C04750=3783,34311,-25890,658,-28447,-2203
C04751=3764,34294,-25911,661,-28441,-2195
C04752=3742,34281,-25927,664,-28436,-2187
C04753=3760,34297,-25907,662,-28442,-2194
C04754=3779,34307,-25895,659,-28446,-2201
C04755=3789,34330,-25867,657,-28455,-2205
C04756=3806,34351,-25841,655,-28463,-2211
C04757=3823,34373,-25815,652,-28471,-2218
C04758=3840,34394,-25789,650,-28479,-2225
C04759=3857,34415,-25763,647,-28487,-2231
C04760=3874,34437,-25737,645,-28495,-2238
C04761=3889,34459,-25710,642,-28504,-2243
C04762=3900,34481,-25683,641,-28512,-2248
C04763=3910,34504,-25655,639,-28521,-2251
C04764=3920,34527,-25627,637,-28530,-2255
C04765=3929,34550,-25599,636,-28538,-2259
C04766=3939,34574,-25571,634,-28547,-2263
C04767=3949,34597,-25543,633,-28556,-2266
C04768=3958,34620,-25514,631,-28565,-2270
C04769=3955,34646,-25483,632,-28574,-2269
C04770=3962,34670,-25454,630,-28583,-2271
C04771=3970,34693,-25425,629,-28592,-2274
C04772=3969,34719,-25394,629,-28602,-2273
C04773=3974,34743,-25364,628,-28611,-2275
C04774=3971,34770,-25333,628,-28621,-2274
C04775=3968,34796,-25301,629,-28630,-2273
C04776=3965,34822,-25269,629,-28640,-2271
C04777=3956,34845,-25241,630,-28648,-2268
C04778=3948,34868,-25213,631,-28657,-2265
C04779=3938,34890,-25187,632,-28665,-2260
C04780=3925,34911,-25162,634,-28673,-2255
C04781=3913,34932,-25137,635,-28680,-2251
C04782=3920,34941,-25125,634,-28684,-2253
C04783=3935,34922,-25149,632,-28677,-2259
C04784=3946,34901,-25174,631,-28669,-2264
C04785=3958,34880,-25200,629,-28661,-2268
C04786=3970,34859,-25225,628,-28654,-2273
C04787=3973,34832,-25257,628,-28644,-2275
C04788=3985,34812,-25282,626,-28636,-2279
C04789=3988,34785,-25313,626,-28627,-2281
C04790=3991,34759,-25345,626,-28617,-2282
C04791=3984,34735,-25374,627,-28608,-2279
C04792=3987,34709,-25406,627,-28598,-2281
C04793=3987,34709,-24006,627,-28598,-2281
C04794=3534,35026,-21027,687,-28710,-2102
C04795=3534,35026,-25027,687,-28710,-2102
C04796=3539,35031,-25020,687,-28712,-2103
C04797=3543,35037,-25013,686,-28714,-2105
C04798=3542,35044,-25005,686,-28717,-2105
C04799=3545,35050,-24998,686,-28719,-2106
C04800=3549,35055,-24991,685,-28721,-2107
C04801=3554,35061,-24984,684,-28724,-2109
C04802=3558,35067,-24977,684,-28726,-2111
C04803=3565,35069,-24975,683,-28727,-2113
C04804=3571,35071,-24971,682,-28728,-2115
C04805=3575,35077,-24964,681,-28730,-2117
C04806=3579,35083,-24958,681,-28732,-2119
C04807=3584,35088,-24951,680,-28734,-2121
C04808=3589,35091,-24947,679,-28735,-2123
C04809=3596,35092,-24946,678,-28736,-2125
C04810=3603,35093,-24944,677,-28736,-2128
C04811=3610,35095,-24943,676,-28737,-2131
C04812=3616,35097,-24939,675,-28738,-2133
C04813=3621,35103,-24932,675,-28740,-2135
C04814=3620,35108,-24927,675,-28742,-2135
C04815=3615,35112,-24922,675,-28743,-2133
C04816=3609,35116,-24917,676,-28745,-2130
C04817=3604,35120,-24912,677,-28746,-2128
C04818=3598,35121,-24911,678,-28747,-2126
C04819=3591,35120,-24912,679,-28746,-2123
C04820=3584,35119,-24913,680,-28746,-2120
C04821=3577,35118,-24914,681,-28745,-2118
C04822=3570,35117,-24916,682,-28745,-2115
C04823=3563,35116,-24917,683,-28744,-2112
C04824=3556,35115,-24918,684,-28744,-2109
C04825=3549,35114,-24920,685,-28743,-2107
C04826=3542,35113,-24921,686,-28743,-2104
C04827=3535,35112,-24922,687,-28742,-2101
C04828=3528,35111,-24924,688,-28742,-2099
C04829=3521,35110,-24925,689,-28741,-2096
C04830=3515,35108,-24928,689,-28740,-2093
C04831=3511,35102,-24935,690,-28738,-2092
C04832=3505,35098,-24940,691,-28737,-2090
C04833=3498,35097,-24941,692,-28736,-2087
C04834=3491,35096,-24942,693,-28736,-2084
C04835=3484,35095,-24944,694,-28735,-2082
C04836=3477,35094,-24945,695,-28735,-2079
C04837=3471,35093,-24946,696,-28734,-2076
C04838=3466,35088,-24952,696,-28732,-2074
C04839=3461,35082,-24959,697,-28730,-2073
C04840=3462,35076,-24967,697,-28728,-2073
C04841=3462,35069,-24976,697,-28725,-2073
C04842=3463,35062,-24984,697,-28723,-2073
C04843=3464,35055,-24992,697,-28720,-2074
C04844=3468,35050,-24998,696,-28719,-2075
C04845=3474,35046,-25003,696,-28717,-2078
C04846=3479,35042,-25008,695,-28716,-2080
C04847=3485,35038,-25013,694,-28714,-2082
C04848=3490,35034,-25018,693,-28713,-2084
C04849=3496,35030,-25023,693,-28711,-2086
C04850=3501,35026,-25028,692,-28710,-2088
C04851=3507,35022,-25032,691,-28708,-2091
C04852=3514,35023,-25031,690,-28709,-2093
C04853=3520,35024,-25029,689,-28709,-2096
C04854=3527,35025,-25028,688,-28710,-2099
C04855=3534,35026,-25027,687,-28710,-2102
C04856=3534,35026,-23627,687,-28710,-2102
C04857=3901,34041,-22216,644,-28348,-2250
C04858=3901,34041,-26216,644,-28348,-2250
C04859=3933,34017,-26245,639,-28340,-2263
C04860=3959,33989,-26278,636,-28330,-2273
C04861=3985,33961,-26312,632,-28319,-2284
C04862=4016,33935,-26343,628,-28310,-2296
C04863=4038,33905,-26380,626,-28299,-2304
C04864=4064,33877,-26413,622,-28289,-2315
C04865=4090,33849,-26447,619,-28279,-2325
C04866=4116,33821,-26481,615,-28269,-2336
C04867=4136,33789,-26519,613,-28257,-2343
C04868=4162,33761,-26553,609,-28247,-2354
C04869=4187,33732,-26588,606,-28237,-2364
C04870=4210,33702,-26623,603,-28226,-2373
C04871=4234,33673,-26659,599,-28215,-2382
C04872=4257,33643,-26695,597,-28204,-2391
C04873=4281,33613,-26731,593,-28193,-2401
C04874=4300,33582,-26769,591,-28182,-2409
C04875=4320,33550,-26807,588,-28170,-2417
C04876=4341,33518,-26845,586,-28159,-2425
C04877=4364,33489,-26881,582,-28148,-2434
C04878=4386,33458,-26918,579,-28137,-2443
C04879=4406,33426,-26956,577,-28125,-2451
C04880=4425,33394,-26995,574,-28113,-2458
C04881=4446,33363,-27033,572,-28102,-2467
C04882=4462,33329,-27074,570,-28089,-2473
C04883=4486,33299,-27110,566,-28079,-2482
C04884=4500,33264,-27152,565,-28066,-2488
C04885=4519,33232,-27191,562,-28054,-2496
C04886=4538,33199,-27230,560,-28042,-2503
C04887=4553,33165,-27272,558,-28029,-2509
C04888=4555,33137,-27306,558,-28019,-2510
C04889=4535,33169,-27267,560,-28031,-2502
C04890=4517,33202,-27227,563,-28043,-2495
C04891=4502,33236,-27186,565,-28055,-2489
C04892=4480,33267,-27149,568,-28066,-2480
C04893=4456,33297,-27113,571,-28077,-2471
C04894=4442,33332,-27071,573,-28090,-2465
C04895=4419,33361,-27035,576,-28101,-2456
C04896=4395,33391,-26999,579,-28112,-2447
C04897=4381,33426,-26956,580,-28125,-2441
C04898=4358,33456,-25521,584,-28136,-2432
C04899=-41004,59868,4099,4900,-34257,16705
C04900=-41004,59868,1099,4900,-34257,16705
C04901=-41004,64596,1380,5213,-31659,16463
C04902=-41004,59868,1099,4900,-34257,16705
C04903=-41004,59868,9099,4900,-34257,16705
C04904=4358,33456,-22921,584,-28136,-2432
C04905=4358,33456,-26921,584,-28136,-2432
C04906=4336,33487,-26884,586,-28147,-2423
C04907=4316,33518,-26845,589,-28158,-2415
C04908=4296,33550,-26807,592,-28170,-2407
C04909=4274,33581,-26771,595,-28181,-2398
C04910=4251,33610,-26735,598,-28192,-2389
C04911=4230,33642,-26697,600,-28203,-2381
C04912=4204,33670,-26663,604,-28214,-2371
C04913=4184,33702,-26625,606,-28225,-2363
C04914=4158,33730,-26591,610,-28235,-2352
C04915=4135,33759,-26555,613,-28246,-2343
C04916=4112,33789,-26519,616,-28257,-2334
C04917=4088,33819,-26483,619,-28268,-2325
C04918=4065,33849,-26447,622,-28279,-2315
C04919=4040,33877,-26413,625,-28289,-2305
C04920=4014,33905,-26379,629,-28299,-2295
C04921=3988,33933,-26346,632,-28309,-2285
C04922=3962,33961,-26312,636,-28319,-2274
C04923=3935,33990,-26278,639,-28330,-2264
C04924=3909,34018,-26244,643,-28340,-2254
C04925=3901,34041,-26216,644,-28348,-2250
C04926=3901,34041,-24816,644,-28348,-2250
C04927=3701,33792,-22519,674,-28253,-2173
C04928=3701,33792,-26519,674,-28253,-2173
C04929=3740,33763,-26554,669,-28243,-2189
C04930=3773,33730,-26594,664,-28231,-2202
C04931=3812,33701,-26629,659,-28221,-2217
C04932=3839,33664,-26673,655,-28207,-2228
C04933=3871,33631,-26713,651,-28195,-2241
C04934=3897,33594,-26757,648,-28182,-2251
C04935=3929,33561,-26798,644,-28170,-2264
C04936=3957,33524,-26841,640,-28157,-2275
C04937=3983,33488,-26885,636,-28143,-2285
C04938=4009,33451,-26930,633,-28130,-2296
C04939=4035,33414,-26975,630,-28116,-2306
C04940=4062,33377,-27018,626,-28103,-2317
C04941=4089,33341,-27063,623,-28090,-2327
C04942=4109,33300,-27112,620,-28075,-2335
C04943=4135,33263,-27156,617,-28061,-2346
C04944=4156,33223,-27204,614,-28047,-2354
C04945=4180,33185,-27250,611,-28033,-2364
C04946=4204,33147,-27296,608,-28019,-2373
C04947=4229,33109,-27342,604,-28005,-2383
C04948=4255,33072,-27387,601,-27991,-2393
C04949=4282,33035,-27431,597,-27978,-2404
C04950=4308,32999,-27475,594,-27965,-2415
C04951=4335,32962,-27520,590,-27951,-2425
C04952=4362,32925,-27564,587,-27938,-2436
C04953=4389,32888,-27608,583,-27924,-2446
C04954=4415,32852,-27652,580,-27911,-2457
C04955=4442,32815,-27697,576,-27898,-2468
C04956=4462,32774,-27746,574,-27883,-2476
C04957=4461,32750,-27775,574,-27874,-2475
C04958=4436,32788,-27730,577,-27888,-2465
C04959=4412,32826,-27684,580,-27901,-2456
C04960=4387,32864,-27638,584,-27915,-2446
C04961=4360,32901,-27594,587,-27929,-2435
C04962=4333,32937,-27549,591,-27942,-2425
C04963=4304,32973,-27507,595,-27955,-2413
C04964=4280,33011,-27461,598,-27969,-2403
C04965=4253,33048,-27416,601,-27982,-2393
C04966=4226,33084,-27372,605,-27996,-2382
C04967=4200,33121,-27328,608,-28009,-2372
C04968=4173,33158,-27284,612,-28022,-2361
C04969=4153,33198,-27235,615,-28037,-2353
C04970=4127,33235,-27190,618,-28051,-2343
C04971=4107,33276,-27141,621,-28066,-2335
C04972=4080,33312,-27097,624,-28079,-2324
C04973=4060,33353,-27048,627,-28094,-2316
C04974=4034,33390,-27004,630,-28107,-2306
C04975=4004,33424,-26962,634,-28120,-2294
C04976=3980,33462,-26916,637,-28134,-2284
C04977=3955,33500,-26871,640,-28147,-2274
C04978=3922,33533,-26831,645,-28159,-2261
C04979=3896,33570,-26787,648,-28173,-2251
C04980=3865,33604,-26746,652,-28185,-2239
C04981=3836,33639,-26703,656,-28198,-2227
C04982=3808,33675,-26660,660,-28211,-2216
C04983=3775,33708,-26621,664,-28223,-2203
C04984=3738,33739,-26584,669,-28234,-2188
C04985=3699,33768,-26549,674,-28244,-2173
C04986=3660,33797,-26514,680,-28255,-2157
C04987=3658,33810,-26499,680,-28259,-2157
C04988=3701,33792,-26519,674,-28253,-2173
C04989=3701,33792,-25119,674,-28253,-2173
C04990=3330,33582,-22776,728,-28171,-2030
C04991=3330,33582,-26776,728,-28171,-2030
C04992=3394,33535,-26833,719,-28154,-2055
C04993=3460,33494,-26882,710,-28140,-2081
C04994=3517,33443,-26944,703,-28121,-2104
C04995=3581,33396,-27001,694,-28104,-2129
C04996=3635,33342,-27064,687,-28085,-2150
C04997=3690,33289,-27128,680,-28066,-2172
C04998=3740,33234,-27195,673,-28046,-2192
C04999=3785,33175,-27266,667,-28025,-2210
C05000=3829,33116,-27336,661,-28003,-2227
C05001=3875,33058,-27407,655,-27982,-2245
C05002=3921,33000,-27476,649,-27961,-2264
C05003=3968,32942,-27546,643,-27940,-2282
C05004=4014,32884,-27616,637,-27919,-2301
C05005=4060,32826,-27686,631,-27898,-2319
C05006=4098,32764,-27762,626,-27875,-2334
C05007=4144,32706,-27832,620,-27854,-2352
C05008=4188,32646,-27903,614,-27832,-2370
C05009=4233,32587,-27974,608,-27811,-2388
C05010=4275,32527,-28047,602,-27788,-2404
C05011=4322,32469,-28117,596,-27767,-2423
C05012=4362,32407,-28191,591,-27745,-2439
C05013=4408,32349,-28262,585,-27723,-2457
C05014=4454,32290,-28333,578,-27702,-2475
C05015=4506,32235,-28399,571,-27682,-2495
C05016=4558,32180,-28466,564,-27662,-2516
C05017=4611,32125,-28532,557,-27642,-2537
C05018=4663,32070,-28598,550,-27622,-2557
C05019=4716,32015,-28664,543,-27602,-2578
C05020=4775,31964,-28725,535,-27584,-2601
C05021=4803,31910,-28791,531,-27564,-2613
C05022=4751,31965,-28725,538,-27584,-2592
C05023=4691,32016,-28664,546,-27602,-2569
C05024=4639,32071,-28597,553,-27622,-2548
C05025=4586,32125,-28531,561,-27642,-2527
C05026=4528,32177,-28469,569,-27661,-2504
C05027=4480,32235,-28399,575,-27682,-2486
C05028=4429,32290,-28333,582,-27702,-2465
C05029=4383,32349,-28262,588,-27723,-2447
C05030=4339,32408,-28190,594,-27745,-2430
C05031=4293,32466,-28120,600,-27766,-2411
C05032=4254,32529,-28045,605,-27789,-2396
C05033=4208,32587,-27975,611,-27810,-2378
C05034=4164,32646,-27903,617,-27832,-2360
C05035=4119,32705,-27832,623,-27853,-2342
C05036=4077,32766,-27759,629,-27876,-2326
C05037=4031,32824,-27689,635,-27897,-2307
C05038=3984,32882,-27619,641,-27918,-2289
C05039=3939,32940,-27549,647,-27939,-2271
C05040=3901,33003,-27473,652,-27962,-2256
C05041=3855,33061,-27404,658,-27983,-2237
C05042=3809,33119,-27334,664,-28004,-2219
C05043=3761,33176,-27265,670,-28025,-2200
C05044=3716,33234,-27194,676,-28046,-2183
C05045=3661,33287,-27131,684,-28065,-2161
C05046=3608,33341,-27067,691,-28084,-2140
C05047=3551,33392,-27005,698,-28103,-2117
C05048=3493,33444,-26943,706,-28121,-2094
C05049=3429,33491,-26886,715,-28138,-2069
C05050=3366,33539,-26829,723,-28155,-2044
C05051=3330,33582,-26776,728,-28171,-2030
C05052=3330,33582,-25376,728,-28171,-2030
C05053=3223,32799,-23726,750,-27878,-1993
C05054=3223,32799,-27726,750,-27878,-1993
C05055=3252,32786,-27741,746,-27874,-2004
C05056=3276,32766,-27765,743,-27867,-2014
C05057=3297,32744,-27792,740,-27859,-2022
C05058=3323,32724,-27815,737,-27852,-2032
C05059=3350,32705,-27838,733,-27845,-2043
C05060=3374,32685,-27862,730,-27838,-2052
C05061=3395,32663,-27889,727,-27830,-2061
C05062=3422,32643,-27913,723,-27823,-2071
C05063=3448,32624,-27936,720,-27816,-2081
C05064=3468,32601,-27964,717,-27808,-2089
C05065=3494,32581,-27987,714,-27801,-2100
C05066=3520,32562,-28010,710,-27794,-2110
C05067=3540,32539,-28038,707,-27785,-2118
C05068=3566,32519,-28061,704,-27778,-2128
C05069=3593,32500,-28085,700,-27771,-2138
C05070=3619,32481,-28108,697,-27765,-2149
C05071=3639,32458,-28136,694,-27756,-2157
C05072=3665,32438,-28159,690,-27749,-2167
C05073=3691,32419,-28182,687,-27742,-2177
C05074=3718,32400,-26805,683,-27735,-2188
C05075=-41004,59868,4099,4900,-34257,16705
C05076=-41004,59868,1099,4900,-34257,16705
C05077=-41004,64596,1380,5213,-31659,16463
C05078=-41004,59868,1099,4900,-34257,16705
C05079=-41004,59868,9099,4900,-34257,16705
C05080=3718,32400,-24205,683,-27735,-2188
C05081=3718,32400,-28205,683,-27735,-2188
C05082=3744,32380,-28229,679,-27729,-2198
C05083=3771,32361,-28252,676,-27722,-2209
C05084=3797,32341,-28275,672,-27715,-2219
C05085=3817,32318,-28303,670,-27706,-2227
C05086=3844,32299,-28326,666,-27699,-2237
C05087=3872,32287,-28341,662,-27695,-2249
C05088=3899,32267,-28364,658,-27688,-2259
C05089=3926,32251,-28384,654,-27682,-2270
C05090=3954,32236,-28402,651,-27677,-2281
C05091=3946,32225,-28415,652,-27673,-2278
C05092=3918,32240,-28397,656,-27678,-2267
C05093=3890,32256,-28377,660,-27684,-2256
C05094=3861,32269,-28363,664,-27688,-2245
C05095=3835,32288,-28339,667,-27695,-2234
C05096=3808,32307,-28316,671,-27702,-2224
C05097=3784,32322,-28299,674,-27707,-2214
C05098=3760,32343,-28274,678,-27715,-2205
C05099=3733,32362,-28250,681,-27722,-2194
C05100=3707,32381,-28227,685,-27729,-2184
C05101=3680,32401,-28204,688,-27736,-2173
C05102=3654,32420,-28181,692,-27742,-2163
C05103=3628,32440,-28158,696,-27749,-2152
C05104=3601,32459,-28134,699,-27756,-2142
C05105=3582,32482,-28106,702,-27765,-2134
C05106=3555,32501,-28083,706,-27772,-2124
C05107=3529,32521,-28060,709,-27779,-2114
C05108=3502,32540,-28037,713,-27785,-2103
C05109=3483,32563,-28009,715,-27794,-2095
C05110=3457,32583,-27986,719,-27801,-2085
C05111=3437,32606,-27958,721,-27809,-2077
C05112=3411,32625,-27935,725,-27816,-2067
C05113=3384,32644,-27911,729,-27823,-2056
C05114=3365,32668,-27883,731,-27831,-2049
C05115=3339,32687,-27860,735,-27838,-2038
C05116=3312,32706,-27837,738,-27845,-2028
C05117=3293,32730,-27809,741,-27854,-2020
C05118=3267,32749,-27786,744,-27860,-2010
C05119=3246,32771,-27759,747,-27869,-2002
C05120=3221,32791,-27735,751,-27876,-1992
C05121=3223,32799,-27726,750,-27878,-1993
C05122=3223,32799,-26326,750,-27878,-1993
C05123=4368,32765,-23758,587,-27878,-2439
C05124=4368,32765,-27758,587,-27878,-2439
C05125=4392,32738,-27791,584,-27868,-2448
C05126=4406,32705,-27830,582,-27856,-2454
C05127=4423,32674,-27868,580,-27845,-2461
C05128=4441,32644,-27904,578,-27834,-2468
C05129=4457,32612,-27943,576,-27822,-2474
C05130=4477,32583,-27978,573,-27812,-2482
C05131=4495,32553,-28014,571,-27800,-2490
C05132=4517,32524,-28048,568,-27790,-2498
C05133=4538,32496,-28083,565,-27780,-2507
C05134=4556,32465,-28120,562,-27768,-2514
C05135=4578,32437,-28154,559,-27758,-2523
C05136=4600,32408,-28188,557,-27748,-2531
C05137=4618,32378,-28225,554,-27737,-2538
C05138=4639,32349,-28260,551,-27726,-2547
C05139=4661,32321,-28294,548,-27716,-2555
C05140=4679,32291,-28330,546,-27705,-2563
C05141=4700,32262,-28365,543,-27694,-2571
C05142=4723,32234,-28399,540,-27684,-2580
C05143=4741,32204,-28436,538,-27673,-2587
C05144=4761,32174,-28471,535,-27662,-2595
C05145=4784,32147,-28504,532,-27652,-2604
C05146=4803,32116,-28541,529,-27641,-2612
C05147=4823,32087,-28577,527,-27630,-2619
C05148=4846,32059,-28610,524,-27620,-2629
C05149=4860,32027,-28649,522,-27608,-2634
C05150=4883,31999,-28683,519,-27598,-2643
C05151=4898,31966,-28722,517,-27586,-2649
C05152=4920,31938,-28756,514,-27575,-2658
C05153=4936,31906,-28794,512,-27564,-2664
C05154=4950,31874,-28834,510,-27552,-2670
C05155=4927,31901,-28801,513,-27562,-2661
C05156=4912,31934,-28761,515,-27574,-2655
C05157=4889,31961,-28728,518,-27584,-2646
C05158=4870,31991,-28692,521,-27595,-2638
C05159=4851,32021,-28656,523,-27606,-2631
C05160=4827,32049,-28623,526,-27616,-2621
C05161=4808,32078,-28587,529,-27627,-2614
C05162=4789,32109,-28550,531,-27638,-2606
C05163=4766,32136,-28517,535,-27648,-2597
C05164=4746,32166,-28481,537,-27659,-2589
C05165=4728,32196,-28445,540,-27670,-2582
C05166=4705,32224,-28411,543,-27680,-2573
C05167=4684,32253,-28376,546,-27691,-2565
C05168=4666,32283,-28340,548,-27702,-2557
C05169=4644,32311,-28306,551,-27712,-2549
C05170=4623,32340,-28271,554,-27722,-2540
C05171=4604,32370,-28234,556,-27734,-2533
C05172=4583,32399,-28200,559,-27744,-2524
C05173=4561,32427,-28166,562,-27754,-2516
C05174=4543,32458,-28129,564,-27766,-2509
C05175=4522,32486,-28094,567,-27776,-2500
C05176=4500,32515,-28060,570,-27786,-2492
C05177=4482,32545,-28024,572,-27797,-2485
C05178=4461,32574,-27989,575,-27808,-2476
C05179=4439,32602,-27955,578,-27818,-2468
C05180=4424,32634,-27916,580,-27830,-2462
C05181=4409,32667,-27877,582,-27842,-2456
C05182=4391,32697,-27840,584,-27853,-2448
C05183=4373,32727,-27804,587,-27864,-2441
C05184=4368,32765,-27758,587,-27878,-2439
C05185=4368,32765,-26358,587,-27878,-2439
C05186=4624,32810,-23702,550,-27898,-2539
C05187=4624,32810,-27702,550,-27898,-2539
C05188=4618,32864,-27636,551,-27918,-2536
C05189=4611,32919,-27570,551,-27938,-2533
C05190=4605,32973,-27504,552,-27958,-2530
C05191=4598,33027,-27438,552,-27978,-2528
C05192=4592,33082,-27373,553,-27999,-2525
C05193=4604,33118,-27328,551,-28012,-2530
C05194=4623,33071,-27385,549,-27995,-2537
C05195=4630,33017,-27451,548,-27975,-2540
C05196=4636,32962,-27517,547,-27955,-2543
C05197=4643,32908,-27583,547,-27934,-2545
C05198=4649,32854,-27648,546,-27914,-2548
C05199=4665,32805,-27708,544,-27896,-2555
C05200=4680,32755,-27768,543,-27878,-2561
C05201=4688,32701,-27833,542,-27858,-2564
C05202=4710,32656,-27888,539,-27841,-2573
C05203=4729,32609,-27945,537,-27824,-2580
C05204=4747,32560,-28003,534,-27806,-2588
C05205=4770,32516,-28057,531,-27790,-2597
C05206=4796,32472,-28110,528,-27773,-2607
C05207=4822,32429,-28162,525,-27757,-2617
C05208=4847,32385,-28215,521,-27741,-2628
C05209=4879,32345,-28263,517,-27727,-2640
C05210=4904,32301,-28316,514,-27711,-2650
C05211=4930,32257,-28369,510,-27695,-2660
C05212=4959,32216,-28419,506,-27679,-2672
C05213=4987,32173,-28470,502,-27664,-2683
C05214=5019,32133,-28519,498,-27649,-2696
C05215=5046,32090,-28571,495,-27633,-2706
C05216=5072,32047,-28624,491,-27617,-2716
C05217=5102,32006,-28673,487,-27602,-2728
C05218=5133,31965,-28722,483,-27587,-2740
C05219=5159,31921,-28775,479,-27571,-2751
C05220=5185,31877,-28828,476,-27555,-2761
C05221=5210,31834,-28881,473,-27539,-2771
C05222=5237,31790,-28933,469,-27523,-2782
C05223=5240,31763,-28967,469,-27513,-2783
C05224=5214,31806,-28914,472,-27529,-2773
C05225=5178,31844,-28868,477,-27543,-2759
C05226=5150,31886,-28817,481,-27558,-2747
C05227=5117,31926,-28769,485,-27573,-2735
C05228=5091,31970,-28716,489,-27589,-2724
C05229=5060,32010,-28668,493,-27604,-2712
C05230=5034,32054,-28615,497,-27620,-2702
C05231=5002,32094,-28566,501,-27634,-2689
C05232=4977,32138,-28514,504,-27651,-2679
C05233=4945,32178,-28465,509,-27665,-2666
C05234=4918,32221,-28413,512,-27681,-2656
C05235=4887,32262,-28364,516,-27696,-2644
C05236=4862,32306,-28311,520,-27712,-2634
C05237=4832,32347,-28262,524,-27727,-2622
C05238=4806,32390,-28209,527,-27743,-2611
C05239=4780,32434,-28156,530,-27759,-2601
C05240=4755,32477,-28104,534,-27775,-2591
C05241=4729,32521,-28051,537,-27791,-2581
C05242=4711,32569,-27993,539,-27809,-2574
C05243=4688,32614,-27939,542,-27825,-2564
C05244=4672,32663,-27880,544,-27843,-2558
C05245=4656,32712,-27820,546,-27861,-2552
C05246=4640,32761,-27761,548,-27880,-2545
C05247=4624,32810,-26302,550,-27898,-2539
C05248=-41004,59868,4099,4900,-34257,16705
C05249=-41004,59868,1099,4900,-34257,16705
C05250=-41004,64596,1380,5213,-31659,16463
C05251=-41004,59868,1099,4900,-34257,16705
C05252=-41004,59868,9099,4900,-34257,16705
C05253=4624,32810,-23702,550,-27898,-2539
C05254=4624,32810,-27702,550,-27898,-2539
C05255=4624,32810,-26302,550,-27898,-2539
C05256=4804,32836,-23668,524,-27909,-2609
C05257=4804,32836,-27668,524,-27909,-2609
C05258=4799,32856,-27644,525,-27917,-2607
C05259=4787,32872,-27625,526,-27923,-2602
C05260=4778,32890,-27604,528,-27929,-2598
C05261=4773,32909,-27580,528,-27936,-2596
C05262=4761,32925,-27561,530,-27942,-2591
C05263=4758,32947,-27535,530,-27950,-2590
C05264=4770,32931,-27554,528,-27944,-2595
C05265=4782,32915,-27573,527,-27938,-2600
C05266=4794,32899,-27592,525,-27933,-2605
C05267=4802,32881,-27614,524,-27926,-2608
C05268=4809,32862,-27637,523,-27919,-2610
C05269=4821,32846,-27657,522,-27913,-2615
C05270=4833,32830,-27676,520,-27907,-2620
C05271=4845,32814,-27695,519,-27902,-2625
C05272=4850,32794,-27719,518,-27894,-2627
C05273=4861,32778,-27739,516,-27888,-2631
C05274=4872,32761,-27758,515,-27882,-2636
C05275=4884,32745,-27778,514,-27876,-2640
C05276=4896,32729,-27797,512,-27870,-2645
C05277=4908,32713,-27817,510,-27865,-2650
C05278=4920,32697,-27836,509,-27859,-2654
C05279=4932,32681,-27855,507,-27853,-2659
C05280=4944,32666,-27874,505,-27847,-2664
C05281=4956,32650,-27893,504,-27841,-2669
C05282=4967,32633,-27913,502,-27835,-2673
C05283=4978,32617,-27933,501,-27829,-2677
C05284=4989,32600,-27953,499,-27823,-2682
C05285=5000,32584,-27973,498,-27817,-2686
C05286=5011,32567,-27993,496,-27811,-2691
C05287=5022,32551,-28013,495,-27805,-2695
C05288=5033,32534,-28033,493,-27799,-2699
C05289=5043,32517,-28053,492,-27793,-2703
C05290=5055,32501,-28073,491,-27787,-2708
C05291=5067,32485,-28092,489,-27781,-2712
C05292=5078,32468,-28112,488,-27775,-2717
C05293=5082,32448,-28137,487,-27767,-2719
C05294=5070,32464,-28118,489,-27773,-2714
C05295=5058,32480,-28098,490,-27779,-2709
C05296=5046,32496,-28079,492,-27785,-2704
C05297=5034,32512,-28060,494,-27791,-2699
C05298=5020,32527,-28042,495,-27796,-2694
C05299=5009,32543,-28022,497,-27802,-2690
C05300=4997,32559,-28002,498,-27808,-2685
C05301=4985,32575,-27983,500,-27814,-2680
C05302=4973,32591,-27964,502,-27820,-2676
C05303=4961,32607,-27945,503,-27825,-2671
C05304=4949,32623,-27926,505,-27831,-2666
C05305=4937,32639,-27906,507,-27837,-2661
C05306=4925,32655,-27887,508,-27843,-2657
C05307=4914,32671,-27867,510,-27849,-2652
C05308=4903,32688,-27847,511,-27855,-2648
C05309=4892,32704,-27827,513,-27861,-2643
C05310=4881,32721,-27808,514,-27867,-2639
C05311=4870,32737,-27788,516,-27873,-2635
C05312=4859,32754,-27768,517,-27879,-2630
C05313=4848,32770,-27748,518,-27885,-2626
C05314=4837,32787,-27728,520,-27891,-2622
C05315=4826,32803,-27708,521,-27897,-2617
C05316=4815,32820,-27688,523,-27903,-2613
C05317=4804,32836,-27668,524,-27909,-2609
C05318=4804,32836,-26268,524,-27909,-2609
C05319=5196,32623,-23924,469,-27834,-2762
C05320=5196,32623,-27924,469,-27834,-2762
C05321=5213,32611,-27938,467,-27830,-2769
C05322=5225,32597,-27955,466,-27824,-2774
C05323=5239,32584,-27971,464,-27820,-2779
C05324=5255,32572,-27985,461,-27816,-2785
C05325=5265,32557,-28004,460,-27810,-2789
C05326=5281,32545,-28018,458,-27806,-2796
C05327=5291,32530,-28036,457,-27800,-2799
C05328=5306,32518,-28051,454,-27796,-2805
C05329=5317,32503,-28069,453,-27790,-2810
C05330=5333,32491,-28083,451,-27786,-2816
C05331=5343,32476,-28102,449,-27780,-2820
C05332=5359,32464,-28116,447,-27776,-2826
C05333=5375,32452,-28130,445,-27772,-2833
C05334=5385,32437,-28148,444,-27766,-2836
C05335=5401,32425,-28162,441,-27762,-2843
C05336=5418,32414,-28176,439,-27758,-2849
C05337=5428,32398,-28195,438,-27752,-2853
C05338=5444,32387,-28209,435,-27748,-2860
C05339=5460,32375,-28223,433,-27744,-2866
C05340=5470,32360,-28242,432,-27738,-2870
C05341=5486,32348,-28256,429,-27734,-2876
C05342=5503,32336,-28270,427,-27730,-2883
C05343=5514,32322,-28287,426,-27724,-2887
C05344=5529,32309,-28302,424,-27720,-2893
C05345=5546,32298,-28316,421,-27716,-2899
C05346=5560,32284,-28332,419,-27711,-2905
C05347=5572,32270,-28349,418,-27706,-2910
C05348=5588,32259,-28363,415,-27702,-2916
C05349=5598,32243,-28382,414,-27696,-2920
C05350=5596,32236,-28391,414,-27693,-2919
C05351=5580,32248,-28377,417,-27697,-2913
C05352=5564,32259,-28363,419,-27701,-2907
C05353=5547,32271,-28349,421,-27706,-2900
C05354=5537,32286,-28330,422,-27711,-2896
C05355=5521,32298,-28316,425,-27716,-2890
C05356=5505,32310,-28302,427,-27720,-2883
C05357=5488,32321,-28288,429,-27724,-2877
C05358=5478,32337,-28269,431,-27730,-2873
C05359=5462,32348,-28255,433,-27734,-2867
C05360=5446,32360,-28241,435,-27738,-2860
C05361=5436,32375,-28223,437,-27744,-2856
C05362=5419,32387,-28209,439,-27748,-2850
C05363=5403,32399,-28195,441,-27752,-2844
C05364=5390,32412,-28178,443,-27757,-2839
C05365=5377,32426,-28162,445,-27762,-2833
C05366=5361,32437,-28148,447,-27766,-2827
C05367=5345,32450,-28133,449,-27770,-2821
C05368=5335,32464,-28115,451,-27776,-2817
C05369=5318,32476,-28101,453,-27780,-2810
C05370=5308,32492,-28083,454,-27786,-2806
C05371=5292,32503,-28069,456,-27790,-2800
C05372=5282,32519,-28050,458,-27796,-2796
C05373=5266,32530,-28036,460,-27800,-2790
C05374=5256,32546,-28017,461,-27806,-2786
C05375=5240,32557,-28003,464,-27810,-2780
C05376=5230,32573,-27985,465,-27815,-2776
C05377=5216,32586,-27969,467,-27820,-2770
C05378=5205,32600,-27952,468,-27825,-2766
C05379=5195,32615,-27933,470,-27831,-2762
C05380=5196,32623,-27924,469,-27834,-2762
C05381=5196,32623,-26524,469,-27834,-2762
C05382=5186,32229,-24402,473,-27686,-2760
C05383=5186,32229,-28402,473,-27686,-2760
C05384=5192,32217,-28416,473,-27682,-2762
C05385=5194,32203,-28433,472,-27677,-2763
C05386=5196,32189,-28450,472,-27672,-2764
C05387=5200,32176,-28466,472,-27667,-2766
C05388=5209,32166,-28478,471,-27663,-2769
C05389=5211,32152,-28495,470,-27658,-2770
C05390=5213,32138,-28512,470,-27653,-2771
C05391=5214,32124,-28529,470,-27648,-2771
C05392=5219,32111,-28544,470,-27643,-2773
C05393=5228,32101,-28557,468,-27639,-2777
C05394=5229,32087,-28574,468,-27634,-2777
C05395=5234,32075,-28589,468,-27629,-2779
C05396=5242,32064,-28601,466,-27626,-2783
C05397=5244,32050,-28619,466,-27620,-2783
C05398=5250,32038,-28633,466,-27616,-2786
C05399=5257,32027,-28646,464,-27612,-2789
C05400=5259,32013,-28663,464,-27607,-2789
C05401=5265,32001,-28677,463,-27602,-2792
C05402=5272,31990,-28691,463,-27598,-2794
C05403=5274,31976,-28708,462,-27593,-2795
C05404=5281,31965,-28722,461,-27589,-2798
C05405=5287,31953,-28736,461,-27585,-2800
C05406=5289,31939,-28753,460,-27579,-2801
C05407=5291,31925,-28770,460,-27574,-2802
C05408=5301,31916,-28781,459,-27571,-2806
C05409=5304,31902,-28797,459,-27566,-2807
C05410=5306,31888,-28815,458,-27560,-2808
C05411=5307,31874,-28832,458,-27555,-2809
C05412=5315,31863,-28845,457,-27551,-2812
C05413=5309,31859,-28850,458,-27550,-2809
C05414=5298,31868,-28839,460,-27553,-2805
C05415=5296,31882,-28822,460,-27558,-2804
C05416=5294,31896,-28805,460,-27563,-2803
C05417=5283,31905,-28794,462,-27566,-2799
C05418=5281,31919,-28777,462,-27572,-2798
C05419=5278,31932,-28761,462,-27577,-2797
C05420=5268,31942,-28750,463,-27580,-2793
C05421=5266,31956,-28733,464,-27585,-2792
C05422=5263,31969,-28717,464,-27590,-2791
C05423=5253,31979,-27305,465,-27594,-2787
C05424=-41004,59868,4099,4900,-34257,16705
C05425=-41004,59868,1099,4900,-34257,16705
C05426=-41004,64596,1380,5213,-31659,16463
C05427=-41004,59868,1099,4900,-34257,16705
C05428=-41004,59868,9099,4900,-34257,16705
C05429=5253,31979,-24705,465,-27594,-2787
C05430=5253,31979,-28705,465,-27594,-2787
C05431=5251,31993,-28688,466,-27599,-2786
C05432=5250,32007,-28671,466,-27604,-2786
C05433=5242,32018,-28658,467,-27608,-2783
C05434=5237,32030,-28643,467,-27613,-2780
C05435=5235,32044,-28626,468,-27618,-2780
C05436=5227,32054,-28613,469,-27622,-2777
C05437=5222,32067,-28598,469,-27626,-2775
C05438=5220,32081,-28581,470,-27632,-2774
C05439=5211,32091,-28569,471,-27635,-2770
C05440=5207,32104,-28554,471,-27640,-2769
C05441=5205,32118,-28537,471,-27645,-2768
C05442=5203,32132,-28520,472,-27650,-2767
C05443=5201,32146,-28502,472,-27656,-2766
C05444=5200,32160,-28485,472,-27661,-2766
C05445=5198,32174,-28468,472,-27666,-2765
C05446=5189,32184,-28456,473,-27670,-2761
C05447=5185,32197,-28441,474,-27675,-2760
C05448=5183,32211,-28423,474,-27680,-2759
C05449=5181,32225,-28406,474,-27685,-2758
C05450=5186,32229,-28402,473,-27686,-2760
C05451=5186,32229,-27002,473,-27686,-2760
C05452=5354,32144,-24503,450,-27657,-2826
C05453=5354,32144,-28503,450,-27657,-2826
C05454=5359,32149,-28498,449,-27658,-2827
C05455=5365,32136,-28513,448,-27654,-2830
C05456=5371,32123,-28529,448,-27649,-2832
C05457=5379,32112,-28543,446,-27645,-2835
C05458=5389,32101,-28555,445,-27641,-2839
C05459=5392,32087,-28573,445,-27636,-2841
C05460=5394,32072,-28591,444,-27630,-2841
C05461=5400,32059,-28606,444,-27625,-2844
C05462=5407,32048,-28620,443,-27621,-2847
C05463=5409,32033,-28639,442,-27615,-2848
C05464=5411,32018,-28657,442,-27610,-2848
C05465=5413,32003,-28675,442,-27604,-2849
C05466=5416,31988,-28692,442,-27599,-2850
C05467=5427,31978,-28705,440,-27595,-2855
C05468=5429,31963,-28723,440,-27590,-2855
C05469=5431,31948,-28741,440,-27584,-2856
C05470=5433,31933,-28759,440,-27578,-2857
C05471=5434,31918,-28777,440,-27573,-2858
C05472=5436,31903,-28795,439,-27567,-2859
C05473=5438,31888,-28813,439,-27562,-2859
C05474=5440,31873,-28831,439,-27556,-2860
C05475=5442,31858,-28850,439,-27551,-2861
C05476=5444,31843,-28868,439,-27545,-2862
C05477=5446,31828,-28886,438,-27539,-2863
C05478=5448,31813,-28904,438,-27534,-2864
C05479=5440,31801,-28919,440,-27529,-2860
C05480=5441,31786,-28937,439,-27524,-2861
C05481=5443,31771,-28956,439,-27518,-2862
C05482=5445,31756,-28974,439,-27512,-2863
C05483=5447,31741,-28992,439,-27507,-2864
C05484=5438,31734,-29000,440,-27504,-2860
C05485=5436,31749,-28982,440,-27510,-2859
C05486=5434,31764,-28964,441,-27515,-2858
C05487=5432,31779,-28946,441,-27521,-2858
C05488=5430,31794,-28928,441,-27526,-2857
C05489=5428,31809,-28910,441,-27532,-2856
C05490=5426,31824,-28892,441,-27538,-2855
C05491=5425,31838,-28874,441,-27543,-2855
C05492=5433,31851,-28858,440,-27548,-2858
C05493=5431,31866,-28840,440,-27553,-2857
C05494=5429,31881,-28822,441,-27559,-2856
C05495=5427,31896,-28804,441,-27565,-2855
C05496=5425,31911,-28786,441,-27570,-2854
C05497=5423,31926,-28768,441,-27576,-2853
C05498=5415,31938,-28753,442,-27580,-2850
C05499=5410,31951,-28738,443,-27585,-2848
C05500=5408,31966,-28720,443,-27590,-2847
C05501=5406,31981,-28702,443,-27596,-2846
C05502=5404,31996,-28683,443,-27601,-2846
C05503=5402,32011,-28665,444,-27607,-2845
C05504=5400,32026,-28647,444,-27613,-2844
C05505=5394,32038,-28632,445,-27617,-2842
C05506=5387,32050,-28617,446,-27622,-2839
C05507=5385,32065,-28599,446,-27627,-2838
C05508=5383,32080,-28581,446,-27633,-2837
C05509=5371,32090,-28569,448,-27636,-2833
C05510=5370,32105,-28551,448,-27642,-2832
C05511=5368,32120,-28533,448,-27647,-2831
C05512=5359,32131,-28519,449,-27652,-2828
C05513=5354,32144,-28503,450,-27657,-2826
C05514=5354,32144,-27103,450,-27657,-2826
C05515=5717,32094,-24562,398,-27641,-2967
C05516=5717,32094,-28562,398,-27641,-2967
C05517=5722,32096,-28559,397,-27642,-2969
C05518=5729,32086,-28571,396,-27638,-2971
C05519=5730,32074,-28586,396,-27634,-2972
C05520=5732,32062,-28601,396,-27629,-2973
C05521=5734,32049,-28616,396,-27625,-2973
C05522=5729,32038,-28630,396,-27621,-2972
C05523=5726,32027,-28643,397,-27616,-2971
C05524=5728,32014,-28659,397,-27612,-2971
C05525=5730,32002,-28674,396,-27607,-2972
C05526=5731,31990,-28689,396,-27602,-2973
C05527=5725,31979,-28701,397,-27598,-2970
C05528=5724,31967,-28716,397,-27594,-2970
C05529=5726,31955,-28731,397,-27589,-2971
C05530=5727,31942,-28746,397,-27585,-2972
C05531=5722,31932,-28759,398,-27581,-2969
C05532=5720,31920,-28773,398,-27576,-2969
C05533=5722,31908,-28788,398,-27572,-2970
C05534=5720,31896,-28802,398,-27567,-2969
C05535=5715,31885,-28815,399,-27563,-2967
C05536=5716,31873,-28830,399,-27559,-2967
C05537=5718,31860,-28845,399,-27554,-2968
C05538=5717,31849,-28860,399,-27550,-2968
C05539=5711,31838,-28872,400,-27545,-2965
C05540=5712,31826,-28888,400,-27541,-2966
C05541=5714,31813,-28903,400,-27536,-2967
C05542=5714,31801,-28917,400,-27532,-2967
C05543=5707,31791,-28930,401,-27528,-2964
C05544=5709,31779,-28945,401,-27523,-2965
C05545=5701,31772,-28952,402,-27521,-2962
C05546=5692,31764,-28963,403,-27517,-2959
C05547=5692,31752,-28977,403,-27513,-2958
C05548=5692,31764,-28963,403,-27517,-2959
C05549=5699,31774,-28950,402,-27521,-2961
C05550=5697,31786,-28935,402,-27526,-2960
C05551=5696,31799,-28920,402,-27531,-2960
C05552=5694,31811,-28905,403,-27535,-2959
C05553=5696,31823,-28891,402,-27540,-2960
C05554=5701,31834,-28878,401,-27544,-2962
C05555=5700,31846,-28863,402,-27548,-2961
C05556=5698,31858,-28848,402,-27553,-2960
C05557=5699,31870,-28834,402,-27557,-2961
C05558=5705,31881,-28821,401,-27561,-2963
C05559=5703,31893,-28806,401,-27566,-2962
C05560=5702,31906,-28791,401,-27571,-2962
C05561=5702,31918,-28776,401,-27575,-2962
C05562=5709,31928,-28763,400,-27579,-2964
C05563=5707,31940,-28748,400,-27584,-2964
C05564=5706,31953,-28733,400,-27588,-2963
C05565=5705,31965,-28719,400,-27593,-2963
C05566=5713,31975,-28706,399,-27597,-2966
C05567=5711,31988,-28691,399,-27601,-2965
C05568=5710,32000,-28676,399,-27606,-2964
C05569=5708,32012,-28661,399,-27611,-2964
C05570=5716,32023,-28649,398,-27614,-2967
C05571=5715,32035,-28634,398,-27619,-2966
C05572=5713,32047,-28619,398,-27624,-2966
C05573=5712,32060,-28604,399,-27628,-2965
C05574=5711,32072,-28589,399,-27633,-2965
C05575=5719,32082,-28577,397,-27637,-2968
C05576=5717,32094,-28562,398,-27641,-2967
C05577=5717,32094,-27162,398,-27641,-2967
C05578=5969,31997,-24678,362,-27607,-3065
C05579=5969,31997,-28678,362,-27607,-3065
C05580=5991,32024,-28646,358,-27617,-3073
C05581=6005,32052,-28611,356,-27628,-3079
C05582=6026,32079,-28579,353,-27638,-3087
C05583=6040,32107,-28544,351,-27649,-3092
C05584=6054,32135,-28510,349,-27660,-3098
C05585=6068,32164,-28475,347,-27671,-3103
C05586=6082,32192,-28441,344,-27681,-3108
C05587=6096,32221,-28406,342,-27692,-3113
C05588=6104,32250,-28370,341,-27703,-3116
C05589=6120,32278,-28336,338,-27714,-3123
C05590=6130,32307,-28301,337,-27725,-3126
C05591=6144,32336,-28266,335,-27736,-3132
C05592=6157,32364,-28231,333,-27746,-3137
C05593=6171,32393,-28197,330,-27757,-3142
C05594=6185,32421,-28162,328,-27768,-3148
C05595=6206,32448,-28130,325,-27778,-3156
C05596=6227,32474,-28097,322,-27788,-3164
C05597=6249,32501,-28065,319,-27799,-3172
C05598=6268,32528,-28032,316,-27809,-3179
C05599=6283,32556,-26598,314,-27819,-3185
C05600=-41004,59868,4099,4900,-34257,16705
C05601=-41004,59868,1099,4900,-34257,16705
C05602=-41004,64596,1380,5213,-31659,16463
C05603=-41004,59868,1099,4900,-34257,16705
C05604=-41004,59868,9099,4900,-34257,16705
C05605=6283,32556,-23998,314,-27819,-3185
C05606=6283,32556,-27998,314,-27819,-3185
C05607=6297,32584,-27963,311,-27830,-3191
C05608=6318,32611,-27931,308,-27840,-3199
C05609=6334,32628,-27910,306,-27847,-3205
C05610=6326,32599,-27946,307,-27836,-3202
C05611=6312,32570,-27981,309,-27825,-3197
C05612=6296,32542,-28014,312,-27815,-3190
C05613=6277,32515,-28048,315,-27804,-3183
C05614=6256,32488,-28080,318,-27794,-3175
C05615=6236,32462,-28113,321,-27784,-3167
C05616=6221,32433,-28147,323,-27773,-3162
C05617=6200,32407,-28179,326,-27763,-3153
C05618=6179,32380,-28212,329,-27753,-3145
C05619=6165,32352,-28246,332,-27742,-3140
C05620=6150,32326,-28278,334,-27732,-3134
C05621=6137,32300,-28309,336,-27722,-3129
C05622=6131,32270,-28346,337,-27711,-3127
C05623=6121,32241,-28381,339,-27700,-3123
C05624=6107,32213,-28416,341,-27689,-3118
C05625=6093,32184,-28450,343,-27678,-3113
C05626=6086,32154,-28487,344,-27667,-3110
C05627=6070,32126,-28521,346,-27657,-3104
C05628=6053,32099,-28554,349,-27646,-3098
C05629=6037,32071,-28588,351,-27635,-3091
C05630=6023,32042,-28623,354,-27625,-3086
C05631=6004,32015,-28656,357,-27614,-3079
C05632=5988,31987,-28690,359,-27604,-3073
C05633=5967,31961,-28722,362,-27594,-3064
C05634=5945,31934,-28755,366,-27583,-3056
C05635=5931,31905,-28789,368,-27573,-3051
C05636=5910,31879,-28822,371,-27563,-3042
C05637=5896,31850,-28856,373,-27552,-3037
C05638=5874,31824,-28889,376,-27542,-3029
C05639=5849,31803,-28914,380,-27534,-3019
C05640=5863,31832,-28879,378,-27544,-3024
C05641=5877,31860,-28845,376,-27555,-3030
C05642=5898,31887,-28812,373,-27565,-3038
C05643=5912,31915,-28778,370,-27576,-3043
C05644=5934,31942,-28745,367,-27586,-3052
C05645=5949,31970,-28711,365,-27597,-3057
C05646=5969,31997,-28678,362,-27607,-3065
C05647=5969,31997,-27278,362,-27607,-3065
C05648=6577,31775,-24944,275,-27530,-3302
C05649=6577,31775,-28944,275,-27530,-3302
C05650=6588,31784,-28933,273,-27533,-3306
C05651=6603,31788,-28928,271,-27535,-3312
C05652=6615,31796,-28918,269,-27538,-3317
C05653=6629,31802,-28911,267,-27540,-3322
C05654=6645,31804,-28908,265,-27541,-3328
C05655=6656,31814,-28896,263,-27545,-3332
C05656=6671,31818,-28892,261,-27546,-3338
C05657=6683,31826,-28882,259,-27550,-3343
C05658=6697,31831,-28876,257,-27552,-3348
C05659=6713,31833,-28873,255,-27553,-3354
C05660=6724,31843,-28860,253,-27556,-3359
C05661=6739,31847,-28856,251,-27558,-3365
C05662=6751,31855,-28846,249,-27561,-3369
C05663=6765,31860,-28840,247,-27563,-3375
C05664=6781,31862,-28837,245,-27564,-3381
C05665=6792,31873,-28824,243,-27568,-3385
C05666=6807,31876,-28821,241,-27569,-3391
C05667=6823,31878,-28818,238,-27570,-3397
C05668=6837,31884,-28810,236,-27573,-3402
C05669=6849,31891,-28801,235,-27576,-3407
C05670=6865,31894,-28798,232,-27577,-3413
C05671=6877,31902,-28789,230,-27580,-3418
C05672=6891,31907,-28782,228,-27582,-3423
C05673=6907,31909,-28779,226,-27583,-3429
C05674=6918,31919,-28767,224,-27587,-3434
C05675=6933,31923,-28763,222,-27588,-3440
C05676=6949,31925,-28760,220,-27589,-3446
C05677=6959,31936,-28746,218,-27593,-3450
C05678=6974,31933,-28750,216,-27592,-3455
C05679=6974,31923,-28762,216,-27588,-3455
C05680=6960,31917,-28769,218,-27586,-3450
C05681=6947,31911,-28777,220,-27584,-3445
C05682=6934,31904,-28786,222,-27581,-3440
C05683=6919,31901,-28789,224,-27580,-3434
C05684=6906,31893,-28799,226,-27577,-3429
C05685=6892,31888,-28805,228,-27575,-3424
C05686=6877,31886,-28808,231,-27574,-3418
C05687=6866,31876,-28820,232,-27570,-3413
C05688=6851,31872,-28824,234,-27568,-3408
C05689=6835,31870,-28827,237,-27567,-3401
C05690=6824,31859,-28841,238,-27563,-3398
C05691=6809,31857,-28844,241,-27562,-3391
C05692=6794,31853,-28849,243,-27561,-3386
C05693=6782,31843,-28860,244,-27557,-3381
C05694=6767,31841,-28863,247,-27556,-3375
C05695=6753,31835,-28870,249,-27554,-3370
C05696=6740,31828,-28879,251,-27551,-3365
C05697=6725,31825,-28882,253,-27550,-3359
C05698=6712,31817,-28892,255,-27547,-3354
C05699=6698,31812,-28899,257,-27544,-3349
C05700=6685,31806,-28906,259,-27542,-3344
C05701=6672,31799,-28915,261,-27539,-3339
C05702=6658,31794,-28921,263,-27537,-3333
C05703=6646,31785,-28931,265,-27534,-3329
C05704=6630,31783,-28934,267,-27533,-3322
C05705=6614,31781,-28937,269,-27532,-3316
C05706=6604,31770,-28950,271,-27528,-3312
C05707=6588,31767,-28954,273,-27527,-3306
C05708=6572,31765,-28957,275,-27526,-3300
C05709=6577,31775,-28944,275,-27530,-3302
C05710=6577,31775,-27544,275,-27530,-3302
C05711=6539,31568,-25195,281,-27452,-3288
C05712=6539,31568,-29195,281,-27452,-3288
C05713=6999,32450,-28122,211,-27787,-3464
C05714=7060,32190,-28437,203,-27690,-3488
C05715=6106,31297,-29527,346,-27347,-3121
C05716=6015,31218,-29623,359,-27316,-3086
C05717=5406,30679,-30280,452,-27110,-2852
C05718=5013,31113,-29756,506,-27269,-2698
C05719=5420,29846,-31289,455,-26799,-2861
C05720=5168,30529,-30462,488,-27052,-2761
C05721=4582,31191,-29664,568,-27294,-2530
C05722=4926,30054,-31039,527,-26873,-2669
C05723=4994,28834,-32517,526,-26419,-2702
C05724=4916,30112,-30969,528,-26895,-2665
C05725=4692,30860,-30064,555,-27172,-2575
C05726=4778,29595,-31596,552,-26701,-2615
C05727=4915,28295,-33169,542,-26218,-2675
C05728=3919,27393,-34263,699,-25878,-2297
C05729=3232,27589,-34028,800,-25947,-2031
C05730=4595,27279,-34399,599,-25839,-2557
C05731=5482,28337,-33117,457,-26237,-2892
C05732=5371,28536,-32877,472,-26311,-2849
C05733=4598,27401,-34252,597,-25884,-2558
C05734=5064,27827,-33736,524,-26045,-2735
C05735=5459,29116,-32174,455,-26527,-2880
C05736=5555,30427,-30585,431,-27017,-2911
C05737=5874,31117,-29746,380,-27278,-3032
C05738=6207,30586,-30388,335,-27082,-3163
C05739=5584,29714,-31449,432,-26751,-2925
C05740=6598,29546,-31649,283,-26695,-3318
C05741=5818,29232,-32032,401,-26573,-3018
C05742=7362,29474,-31734,170,-26673,-3612
C05743=6312,29284,-31967,327,-26596,-3208
C05744=5551,28467,-32960,446,-26286,-2919
C05745=6148,28896,-32438,354,-26450,-3146
C05746=6650,29254,-32003,277,-26587,-3339
C05747=6189,28425,-33010,351,-26274,-3164
C05748=5391,27925,-33617,474,-26083,-2860
C05749=4173,27168,-34535,663,-25796,-2396
C05750=2987,27817,-33752,835,-26030,-1935
C05751=2342,28406,-33042,924,-26244,-1682
C05752=1685,27796,-33780,1029,-26014,-1433
C05753=596,27535,-34098,1195,-25911,-1016
C05754=674,26114,-35812,1203,-25389,-1060
C05755=2286,26334,-35544,957,-25478,-1677
C05756=3902,26565,-35264,710,-25571,-2296
C05757=5518,26796,-34984,463,-25663,-2914
C05758=7133,27027,-34704,217,-25756,-3533
C05759=7903,27809,-33755,96,-26052,-3825
C05760=7326,28876,-32460,178,-26449,-3600
C05761=7718,28990,-32321,119,-26494,-3751
C05762=6918,29697,-31464,235,-26754,-3440
C05763=7107,29587,-31597,207,-26714,-3514
C05764=6858,30033,-31057,242,-26880,-3416
C05765=7533,30170,-30888,141,-26935,-3676
C05766=6855,30666,-30289,239,-27116,-3413
C05767=6881,31053,-29820,234,-27261,-3422
C05768=7239,30568,-30407,183,-27082,-3562
C05769=7049,31307,-29510,208,-27358,-3486
C05770=6393,31164,-29687,304,-27299,-3232
C05771=7271,31843,-28858,173,-27561,-3571
C05772=6539,31568,-27795,281,-27452,-3288
C05773=-41004,59868,4099,4900,-34257,16705
C05774=-41004,59868,1099,4900,-34257,16705
C05775=-41004,64596,1380,5213,-31659,16463
C05776=-41004,59868,1099,4900,-34257,16705
C05777=-41004,59868,9099,4900,-34257,16705
C05778=6539,31568,-25195,281,-27452,-3288
C05779=6539,31568,-29195,281,-27452,-3288
C05780=6539,31568,-27795,281,-27452,-3288
C05781=6861,31558,-25207,234,-27451,-3412
C05782=6861,31558,-29207,234,-27451,-3412
C05783=6862,31571,-29191,234,-27456,-3413
C05784=6874,31579,-29181,232,-27459,-3417
C05785=6885,31587,-29170,231,-27462,-3422
C05786=6898,31592,-29165,229,-27464,-3427
C05787=6911,31598,-29157,227,-27466,-3432
C05788=6923,31605,-29149,225,-27469,-3436
C05789=6937,31609,-29144,223,-27470,-3442
C05790=6948,31618,-29133,221,-27474,-3446
C05791=6960,31625,-29124,220,-27477,-3451
C05792=6972,31631,-29117,218,-27479,-3455
C05793=6982,31642,-29103,216,-27483,-3459
C05794=6991,31653,-29090,215,-27488,-3463
C05795=7005,31652,-29092,213,-27487,-3468
C05796=7019,31648,-29096,211,-27486,-3473
C05797=7034,31650,-29094,209,-27487,-3479
C05798=7049,31652,-29091,207,-27488,-3485
C05799=7062,31646,-29098,205,-27486,-3490
C05800=7076,31646,-29098,203,-27486,-3496
C05801=7091,31649,-29095,200,-27487,-3502
C05802=7106,31651,-29092,198,-27488,-3507
C05803=7121,31653,-29089,196,-27489,-3513
C05804=7137,31655,-29087,194,-27489,-3519
C05805=7152,31657,-29084,192,-27490,-3525
C05806=7167,31660,-29081,189,-27491,-3531
C05807=7182,31662,-29078,187,-27492,-3537
C05808=7196,31665,-29075,185,-27494,-3542
C05809=7206,31675,-29062,183,-27497,-3546
C05810=7221,31677,-29060,181,-27498,-3552
C05811=7237,31679,-29057,179,-27499,-3558
C05812=7250,31676,-29060,177,-27498,-3563
C05813=7248,31671,-29066,177,-27497,-3562
C05814=7238,31661,-29079,179,-27493,-3558
C05815=7224,31658,-29083,181,-27491,-3553
C05816=7208,31656,-29085,183,-27490,-3547
C05817=7193,31654,-29088,185,-27489,-3541
C05818=7182,31646,-29097,187,-27487,-3537
C05819=7169,31641,-29104,189,-27484,-3532
C05820=7154,31638,-29107,191,-27483,-3526
C05821=7139,31636,-29110,193,-27482,-3520
C05822=7124,31634,-29112,196,-27481,-3514
C05823=7108,31632,-29115,198,-27481,-3508
C05824=7093,31630,-29118,200,-27480,-3502
C05825=7078,31627,-29121,202,-27479,-3497
C05826=7063,31625,-29123,205,-27478,-3491
C05827=7050,31629,-29118,206,-27479,-3486
C05828=7036,31631,-29117,209,-27480,-3480
C05829=7022,31632,-29115,211,-27480,-3475
C05830=7008,31636,-29110,212,-27481,-3469
C05831=6997,31628,-29121,214,-27478,-3465
C05832=6984,31623,-29127,216,-27476,-3460
C05833=6975,31611,-29141,217,-27472,-3457
C05834=6965,31601,-29153,219,-27468,-3453
C05835=6953,31594,-29161,221,-27465,-3448
C05836=6940,31588,-29169,223,-27463,-3443
C05837=6926,31584,-29174,225,-27461,-3438
C05838=6916,31575,-29185,226,-27458,-3434
C05839=6900,31573,-29188,228,-27457,-3428
C05840=6891,31562,-29201,230,-27452,-3424
C05841=6876,31560,-29204,232,-27452,-3418
C05842=6861,31558,-29207,234,-27451,-3412
C05843=6861,31558,-27807,234,-27451,-3412
C05844=6959,31491,-25286,220,-27427,-3451
C05845=6959,31491,-29286,220,-27427,-3451
C05846=6970,31497,-29280,219,-27429,-3455
C05847=6979,31504,-29271,217,-27431,-3458
C05848=6989,31509,-29265,216,-27433,-3462
C05849=6998,31517,-29255,215,-27436,-3466
C05850=7008,31521,-29250,213,-27438,-3470
C05851=7017,31529,-29240,212,-27441,-3473
C05852=7024,31539,-29228,211,-27445,-3476
C05853=7032,31548,-29217,209,-27449,-3479
C05854=7041,31555,-29209,208,-27451,-3482
C05855=7051,31561,-29201,207,-27453,-3486
C05856=7059,31570,-29190,205,-27457,-3489
C05857=7067,31578,-29181,204,-27460,-3493
C05858=7078,31583,-29174,203,-27462,-3496
C05859=7085,31593,-29163,201,-27466,-3499
C05860=7093,31600,-29154,200,-27468,-3502
C05861=7103,31593,-29163,199,-27466,-3506
C05862=7113,31586,-29171,197,-27463,-3510
C05863=7104,31583,-29174,199,-27462,-3507
C05864=7097,31574,-29186,200,-27459,-3504
C05865=7089,31564,-29197,201,-27455,-3501
C05866=7078,31560,-29202,203,-27453,-3497
C05867=7070,31551,-29213,204,-27450,-3494
C05868=7063,31542,-29224,205,-27446,-3491
C05869=7052,31537,-29230,207,-27445,-3487
C05870=7043,31529,-29240,208,-27441,-3483
C05871=7036,31520,-29252,209,-27438,-3480
C05872=7026,31514,-29258,210,-27436,-3477
C05873=7017,31507,-29267,212,-27433,-3473
C05874=7006,31502,-29273,213,-27431,-3469
C05875=6998,31494,-29283,215,-27428,-3466
C05876=6987,31490,-29288,216,-27426,-3462
C05877=6979,31482,-29298,217,-27423,-3458
C05878=6968,31477,-29304,219,-27421,-3454
C05879=6955,31475,-29306,221,-27420,-3449
C05880=6948,31466,-29318,222,-27417,-3447
C05881=6936,31463,-29321,224,-27416,-3442
C05882=6925,31459,-29326,225,-27414,-3438
C05883=6917,31451,-29336,227,-27411,-3434
C05884=6904,31449,-29338,228,-27410,-3430
C05885=6892,31447,-29341,230,-27409,-3425
C05886=6879,31445,-29343,232,-27409,-3420
C05887=6867,31443,-29345,234,-27408,-3415
C05888=6854,31442,-29347,236,-27407,-3410
C05889=6842,31440,-29350,238,-27406,-3405
C05890=6829,31438,-29352,239,-27405,-3401
C05891=6817,31436,-29354,241,-27405,-3396
C05892=6815,31448,-29340,241,-27409,-3395
C05893=6819,31456,-29331,241,-27412,-3397
C05894=6831,31457,-29328,239,-27413,-3401
C05895=6844,31459,-29326,237,-27414,-3406
C05896=6856,31461,-29324,235,-27414,-3411
C05897=6869,31463,-29322,234,-27415,-3416
C05898=6881,31465,-29319,232,-27416,-3421
C05899=6894,31466,-29317,230,-27417,-3425
C05900=6906,31468,-29315,228,-27417,-3430
C05901=6919,31470,-29312,226,-27418,-3435
C05902=6931,31472,-29310,224,-27419,-3440
C05903=6940,31479,-29302,223,-27422,-3444
C05904=6950,31484,-29295,222,-27424,-3447
C05905=6959,31491,-29286,220,-27427,-3451
C05906=6959,31491,-27886,220,-27427,-3451
C05907=7088,31159,-25689,203,-27303,-3502
C05908=7088,31159,-29689,203,-27303,-3502
C05909=7116,31163,-29684,199,-27305,-3512
C05910=7141,31157,-29691,195,-27303,-3522
C05911=7166,31151,-29698,191,-27301,-3532
C05912=7189,31140,-29712,188,-27297,-3541
C05913=7214,31131,-29722,184,-27294,-3550
C05914=7238,31123,-29732,181,-27291,-3560
C05915=7261,31108,-29751,178,-27285,-3569
C05916=7283,31093,-29769,174,-27280,-3577
C05917=7298,31073,-29793,172,-27272,-3583
C05918=7311,31053,-29817,171,-27265,-3588
C05919=7323,31032,-29843,169,-27257,-3593
C05920=7329,31007,-29873,168,-27248,-3595
C05921=7333,30981,-29904,168,-27238,-3597
C05922=7344,30959,-29931,166,-27230,-3601
C05923=7350,30935,-29960,165,-27221,-3604
C05924=7354,30910,-29991,165,-27212,-3605
C05925=7358,30884,-30022,164,-27202,-3607
C05926=7362,30859,-30053,164,-27192,-3609
C05927=7368,30834,-30083,163,-27183,-3611
C05928=7380,30813,-30109,161,-27175,-3616
C05929=7384,30787,-30140,161,-27166,-3617
C05930=7388,30761,-30171,160,-27156,-3619
C05931=7381,30738,-30199,161,-27147,-3616
C05932=7374,30715,-30227,163,-27139,-3614
C05933=7356,30700,-30246,165,-27133,-3606
C05934=7357,30724,-30216,165,-27142,-3607
C05935=7367,30747,-30189,164,-27150,-3611
C05936=7368,30771,-30159,163,-27160,-3611
C05937=7368,30792,-30133,163,-27168,-3611
C05938=7359,30815,-30106,164,-27176,-3607
C05939=7355,30841,-30075,165,-27186,-3606
C05940=7351,30866,-30044,165,-27195,-3604
C05941=7337,30887,-30019,167,-27203,-3599
C05942=7333,30912,-29988,168,-27212,-3597
C05943=7329,30938,-29957,168,-27222,-3596
C05944=7325,30964,-29926,169,-27232,-3594
C05945=7321,30989,-29895,169,-27241,-3592
C05946=7308,31009,-29870,171,-27249,-3587
C05947=7304,31035,-29839,172,-27258,-3585
C05948=7289,31055,-28415,174,-27266,-3580
C05949=-41004,59868,4099,4900,-34257,16705
C05950=-41004,59868,1099,4900,-34257,16705
C05951=-41004,64596,1380,5213,-31659,16463
C05952=-41004,59868,1099,4900,-34257,16705
C05953=-41004,59868,9099,4900,-34257,16705
C05954=7289,31055,-25815,174,-27266,-3580
C05955=7289,31055,-29815,174,-27266,-3580
C05956=7274,31074,-29792,176,-27273,-3574
C05957=7251,31089,-29773,179,-27278,-3565
C05958=7229,31104,-29755,182,-27284,-3556
C05959=7206,31119,-29738,186,-27289,-3547
C05960=7181,31125,-29730,189,-27291,-3538
C05961=7156,31131,-29723,193,-27293,-3528
C05962=7133,31144,-29707,196,-27298,-3519
C05963=7107,31146,-29706,200,-27298,-3509
C05964=7084,31144,-29707,203,-27297,-3500
C05965=7063,31129,-29725,207,-27292,-3492
C05966=7037,31123,-29733,210,-27289,-3482
C05967=7009,31119,-29738,215,-27287,-3471
C05968=6981,31115,-29743,219,-27286,-3460
C05969=6954,31115,-29744,223,-27285,-3450
C05970=6955,31130,-29725,222,-27291,-3450
C05971=6983,31134,-29720,218,-27293,-3461
C05972=7010,31138,-29715,214,-27295,-3472
C05973=7038,31142,-29710,210,-27296,-3482
C05974=7066,31146,-29705,206,-27298,-3493
C05975=7088,31159,-29689,203,-27303,-3502
C05976=7088,31159,-28289,203,-27303,-3502
C05977=6957,31046,-25828,222,-27259,-3451
C05978=6957,31046,-29828,222,-27259,-3451
C05979=6973,31021,-29857,220,-27250,-3457
C05980=6990,30998,-29886,218,-27242,-3464
C05981=7010,30976,-29912,215,-27234,-3472
C05982=7039,30965,-29926,211,-27230,-3483
C05983=7068,30953,-29939,207,-27226,-3494
C05984=7096,30940,-29955,203,-27221,-3505
C05985=7124,30924,-29975,199,-27215,-3516
C05986=7147,30903,-30000,195,-27208,-3525
C05987=7171,30883,-30024,192,-27200,-3534
C05988=7185,30858,-30054,190,-27191,-3540
C05989=7199,30833,-30085,188,-27182,-3546
C05990=7211,30806,-30117,186,-27172,-3550
C05991=7218,30777,-30153,185,-27161,-3553
C05992=7224,30747,-30189,185,-27149,-3555
C05993=7237,30721,-30221,183,-27140,-3561
C05994=7252,30696,-30251,181,-27131,-3566
C05995=7271,30673,-30279,178,-27122,-3574
C05996=7291,30651,-30305,175,-27114,-3582
C05997=7318,30633,-30327,171,-27107,-3592
C05998=7347,30622,-30341,167,-27103,-3603
C05999=7378,30617,-30347,162,-27102,-3615
C06000=7373,30606,-30359,163,-27098,-3613
C06001=7340,30601,-30365,168,-27096,-3600
C06002=7312,30617,-30347,172,-27101,-3590
C06003=7283,30631,-30330,176,-27106,-3579
C06004=7263,30653,-30303,179,-27115,-3571
C06005=7243,30675,-30276,182,-27123,-3563
C06006=7230,30701,-30245,184,-27132,-3558
C06007=7216,30726,-30214,186,-27142,-3552
C06008=7203,30752,-30183,188,-27151,-3547
C06009=7197,30782,-30147,188,-27163,-3545
C06010=7190,30812,-30111,189,-27174,-3542
C06011=7178,30838,-30079,191,-27183,-3537
C06012=7163,30863,-30048,193,-27193,-3532
C06013=7136,30882,-30026,197,-27199,-3521
C06014=7109,30900,-30004,201,-27206,-3511
C06015=7083,30918,-29982,205,-27213,-3500
C06016=7056,30936,-29960,208,-27219,-3490
C06017=7029,30955,-29938,212,-27226,-3479
C06018=7007,30970,-29920,216,-27231,-3471
C06019=6980,30988,-29898,219,-27238,-3460
C06020=6959,30973,-29916,222,-27232,-3452
C06021=6953,30944,-29951,224,-27221,-3450
C06022=6957,30914,-29988,223,-27210,-3452
C06023=6962,30883,-30025,222,-27199,-3454
C06024=6975,30857,-30057,221,-27189,-3459
C06025=6988,30831,-30088,219,-27179,-3464
C06026=7001,30805,-30119,217,-27170,-3469
C06027=7015,30785,-30144,215,-27162,-3474
C06028=6992,30795,-30132,218,-27166,-3465
C06029=6972,30817,-30105,221,-27174,-3458
C06030=6958,30843,-30074,223,-27183,-3452
C06031=6953,30873,-30037,224,-27195,-3450
C06032=6949,30904,-30000,224,-27206,-3448
C06033=6944,30934,-29963,225,-27218,-3446
C06034=6947,30963,-29928,224,-27229,-3448
C06035=6945,30993,-29891,224,-27240,-3447
C06036=6941,31024,-29854,225,-27251,-3445
C06037=6936,31055,-29817,225,-27263,-3443
C06038=6957,31046,-29828,222,-27259,-3451
C06039=6957,31046,-28428,222,-27259,-3451
C06040=6526,30749,-26189,287,-27145,-3285
C06041=6526,30749,-30189,287,-27145,-3285
C06042=6549,30725,-30219,284,-27136,-3294
C06043=6558,30695,-30255,283,-27125,-3298
C06044=6556,30662,-30295,283,-27113,-3297
C06045=6532,30647,-30313,287,-27107,-3288
C06046=6494,30642,-30320,292,-27105,-3273
C06047=6456,30636,-30326,298,-27102,-3259
C06048=6423,30622,-30344,303,-27097,-3246
C06049=6385,30617,-30351,308,-27094,-3231
C06050=6400,30638,-30325,306,-27102,-3237
C06051=6433,30652,-30307,301,-27108,-3250
C06052=6471,30658,-30301,296,-27110,-3264
C06053=6507,30666,-30290,290,-27114,-3278
C06054=6530,30694,-30256,287,-27125,-3287
C06055=6522,30727,-30217,288,-27137,-3284
C06056=6491,30748,-30192,292,-27144,-3272
C06057=6457,30754,-30184,297,-27146,-3259
C06058=6421,30756,-30182,302,-27147,-3245
C06059=6386,30760,-30176,308,-27148,-3231
C06060=6348,30755,-30183,313,-27146,-3217
C06061=6313,30760,-30178,318,-27147,-3203
C06062=6276,30754,-30185,324,-27145,-3188
C06063=6238,30749,-30191,329,-27143,-3174
C06064=6200,30743,-30198,335,-27140,-3159
C06065=6162,30738,-30205,341,-27138,-3144
C06066=6124,30732,-30212,346,-27136,-3130
C06067=6086,30727,-30219,352,-27133,-3115
C06068=6048,30721,-30226,357,-27131,-3101
C06069=6016,30707,-30243,362,-27125,-3088
C06070=5978,30701,-30250,368,-27123,-3073
C06071=5940,30696,-30257,373,-27121,-3059
C06072=5908,30682,-30274,378,-27115,-3046
C06073=5870,30676,-30281,384,-27113,-3032
C06074=5837,30662,-30298,389,-27107,-3019
C06075=5800,30656,-30305,394,-27105,-3005
C06076=5767,30642,-30323,399,-27099,-2992
C06077=5729,30637,-30329,405,-27097,-2977
C06078=5709,30643,-30322,408,-27099,-2969
C06079=5742,30656,-30306,403,-27104,-2982
C06080=5773,30672,-30287,398,-27110,-2994
C06081=5806,30686,-30269,393,-27116,-3007
C06082=5844,30691,-30262,387,-27118,-3022
C06083=5882,30697,-30256,382,-27121,-3036
C06084=5914,30711,-30238,377,-27126,-3049
C06085=5952,30717,-30231,371,-27128,-3063
C06086=5984,30731,-30214,367,-27134,-3076
C06087=6022,30736,-30207,361,-27136,-3090
C06088=6060,30742,-30200,355,-27139,-3105
C06089=6098,30747,-30193,350,-27141,-3120
C06090=6136,30753,-30187,344,-27143,-3134
C06091=6174,30758,-30180,339,-27146,-3149
C06092=6211,30764,-30173,333,-27148,-3164
C06093=6244,30778,-30155,328,-27154,-3176
C06094=6279,30774,-30161,323,-27152,-3190
C06095=6317,30779,-30154,318,-27155,-3204
C06096=6352,30775,-30159,313,-27153,-3218
C06097=6389,30780,-30152,307,-27156,-3232
C06098=6424,30776,-30158,302,-27154,-3246
C06099=6459,30771,-30163,297,-27153,-3260
C06100=6493,30763,-30173,292,-27150,-3273
C06101=6526,30749,-30189,287,-27145,-3285
C06102=6526,30749,-28789,287,-27145,-3285
C06103=6602,30476,-26521,277,-27043,-3316
C06104=6602,30476,-30521,277,-27043,-3316
C06105=6649,30482,-30513,270,-27046,-3334
C06106=6696,30489,-30504,263,-27049,-3352
C06107=6743,30496,-30496,257,-27052,-3370
C06108=6789,30503,-30487,250,-27055,-3388
C06109=6836,30509,-30479,243,-27058,-3406
C06110=6880,30506,-30483,236,-27057,-3423
C06111=6927,30513,-30474,229,-27060,-3441
C06112=6974,30520,-30466,222,-27063,-3459
C06113=7016,30509,-30479,216,-27059,-3476
C06114=7027,30489,-30503,215,-27051,-3480
C06115=6980,30482,-30511,222,-27049,-3462
C06116=6939,30494,-30498,228,-27053,-3446
C06117=6892,30489,-30504,235,-27050,-3428
C06118=6845,30482,-30512,241,-27047,-3410
C06119=6801,30485,-30509,248,-27048,-3393
C06120=6754,30478,-30517,255,-27045,-3375
C06121=6707,30472,-30525,262,-27043,-3356
C06122=6661,30465,-30534,269,-27040,-3338
C06123=6614,30458,-30542,276,-27037,-3320
C06124=6567,30451,-29151,283,-27034,-3302
C06125=-41004,59868,4099,4900,-34257,16705
C06126=-41004,59868,1099,4900,-34257,16705
C06127=-41004,64596,1380,5213,-31659,16463
C06128=-41004,59868,1099,4900,-34257,16705
C06129=-41004,59868,9099,4900,-34257,16705
C06130=6567,30451,-26551,283,-27034,-3302
C06131=6567,30451,-30551,283,-27034,-3302
C06132=6520,30445,-30559,290,-27031,-3284
C06133=6473,30438,-30567,296,-27028,-3266
C06134=6432,30422,-30587,303,-27022,-3250
C06135=6385,30415,-30595,310,-27019,-3232
C06136=6338,30409,-30603,317,-27016,-3214
C06137=6291,30402,-30612,323,-27013,-3196
C06138=6244,30395,-30620,330,-27010,-3178
C06139=6203,30380,-30639,337,-27004,-3162
C06140=6156,30373,-30648,344,-27001,-3144
C06141=6109,30366,-30656,350,-26999,-3125
C06142=6062,30359,-30664,357,-26996,-3107
C06143=6015,30352,-30673,364,-26993,-3089
C06144=5971,30356,-30669,371,-26994,-3072
C06145=5924,30349,-30678,378,-26991,-3054
C06146=5878,30342,-30686,385,-26988,-3036
C06147=5831,30335,-30694,392,-26985,-3018
C06148=5787,30338,-30691,398,-26986,-3001
C06149=5743,30342,-30687,404,-26987,-2984
C06150=5699,30345,-30683,411,-26988,-2967
C06151=5686,30356,-30669,413,-26992,-2962
C06152=5731,30359,-30666,406,-26993,-2979
C06153=5775,30355,-30671,400,-26992,-2996
C06154=5819,30353,-30673,393,-26991,-3013
C06155=5866,30360,-30665,386,-26994,-3031
C06156=5913,30366,-30656,379,-26997,-3050
C06157=5957,30363,-30660,373,-26996,-3067
C06158=6004,30370,-30652,366,-26999,-3085
C06159=6050,30377,-30643,359,-27002,-3103
C06160=6097,30383,-30635,352,-27005,-3121
C06161=6144,30390,-30626,345,-27008,-3139
C06162=6186,30406,-30607,339,-27014,-3155
C06163=6232,30413,-30599,332,-27017,-3173
C06164=6279,30419,-30591,325,-27020,-3191
C06165=6326,30426,-30582,318,-27023,-3209
C06166=6373,30433,-30574,311,-27026,-3227
C06167=6414,30448,-30555,305,-27032,-3243
C06168=6461,30455,-30546,298,-27035,-3261
C06169=6508,30462,-30538,291,-27037,-3279
C06170=6555,30469,-30529,284,-27040,-3298
C06171=6602,30476,-30521,277,-27043,-3316
C06172=6602,30476,-29121,277,-27043,-3316
C06173=6752,30236,-26811,256,-26955,-3374
C06174=6752,30236,-30811,256,-26955,-3374
C06175=6782,30243,-30803,252,-26957,-3386
C06176=6814,30248,-30797,247,-26959,-3398
C06177=6840,30261,-30781,243,-26965,-3408
C06178=6872,30266,-30775,239,-26967,-3421
C06179=6893,30287,-30749,235,-26975,-3429
C06180=6918,30301,-30732,232,-26980,-3439
C06181=6944,30316,-30714,228,-26986,-3448
C06182=6963,30339,-30685,225,-26995,-3456
C06183=6986,30357,-30664,221,-27002,-3465
C06184=7006,30381,-30635,218,-27011,-3472
C06185=7030,30389,-30624,215,-27014,-3482
C06186=7030,30366,-30653,215,-27005,-3481
C06187=7010,30343,-30680,218,-26997,-3474
C06188=6987,30324,-30703,221,-26989,-3465
C06189=6964,30307,-30724,225,-26983,-3456
C06190=6937,30294,-30740,229,-26978,-3446
C06191=6913,30278,-30760,232,-26972,-3437
C06192=6891,30259,-30783,236,-26964,-3428
C06193=6865,30245,-30800,240,-26959,-3418
C06194=6839,30232,-30816,244,-26954,-3408
C06195=6807,30227,-30822,248,-26952,-3396
C06196=6775,30223,-30827,253,-26950,-3383
C06197=6749,30210,-30842,257,-26945,-3373
C06198=6717,30205,-30849,262,-26943,-3361
C06199=6686,30200,-30855,266,-26941,-3349
C06200=6654,30197,-30860,271,-26939,-3337
C06201=6631,30192,-30865,275,-26937,-3328
C06202=6609,30172,-30889,278,-26930,-3319
C06203=6597,30147,-30920,280,-26920,-3315
C06204=6585,30122,-30951,282,-26911,-3310
C06205=6565,30098,-30980,285,-26902,-3303
C06206=6542,30080,-31001,288,-26895,-3294
C06207=6514,30069,-31015,292,-26890,-3283
C06208=6487,30057,-31030,296,-26886,-3273
C06209=6456,30052,-31035,301,-26884,-3261
C06210=6424,30047,-31041,306,-26882,-3248
C06211=6395,30053,-31035,310,-26884,-3237
C06212=6366,30058,-31028,314,-26885,-3226
C06213=6337,30064,-31022,319,-26887,-3215
C06214=6310,30074,-31009,323,-26891,-3204
C06215=6282,30084,-30997,327,-26894,-3194
C06216=6290,30105,-30972,325,-26902,-3196
C06217=6317,30094,-30985,321,-26899,-3207
C06218=6345,30084,-30997,317,-26895,-3218
C06219=6372,30074,-31009,313,-26891,-3228
C06220=6402,30071,-31013,309,-26890,-3240
C06221=6431,30068,-31017,305,-26889,-3251
C06222=6463,30072,-31011,300,-26891,-3263
C06223=6495,30077,-31005,295,-26893,-3276
C06224=6521,30090,-30989,291,-26898,-3286
C06225=6545,30107,-30969,288,-26905,-3295
C06226=6559,30131,-30939,285,-26914,-3300
C06227=6577,30156,-30909,283,-26923,-3307
C06228=6588,30181,-30878,281,-26933,-3311
C06229=6608,30205,-30850,278,-26942,-3319
C06230=6630,30213,-30840,275,-26945,-3327
C06231=6661,30216,-30836,270,-26946,-3339
C06232=6693,30220,-30830,265,-26948,-3352
C06233=6724,30225,-30825,261,-26950,-3364
C06234=6752,30236,-30811,256,-26955,-3374
C06235=6752,30236,-29411,256,-26955,-3374
C06236=7130,30197,-26857,201,-26943,-3521
C06237=7130,30197,-30857,201,-26943,-3521
C06238=7142,30196,-30858,199,-26943,-3525
C06239=7153,30191,-30864,197,-26941,-3529
C06240=7165,30189,-30866,196,-26940,-3534
C06241=7176,30185,-30872,194,-26938,-3538
C06242=7187,30183,-30874,192,-26938,-3543
C06243=7199,30179,-30879,191,-26936,-3547
C06244=7210,30176,-30883,189,-26935,-3552
C06245=7220,30169,-30891,188,-26933,-3556
C06246=7231,30164,-30897,186,-26931,-3560
C06247=7243,30162,-30899,184,-26930,-3564
C06248=7253,30155,-30908,183,-26928,-3568
C06249=7264,30150,-30914,181,-26926,-3573
C06250=7276,30148,-30916,179,-26925,-3577
C06251=7287,30143,-30922,178,-26924,-3581
C06252=7299,30141,-30924,176,-26923,-3586
C06253=7310,30137,-30929,174,-26921,-3590
C06254=7322,30135,-30932,173,-26921,-3595
C06255=7333,30131,-30937,171,-26919,-3599
C06256=7346,30133,-30935,169,-26920,-3604
C06257=7359,30135,-30932,167,-26921,-3609
C06258=7369,30128,-30940,166,-26918,-3613
C06259=7382,30128,-30940,164,-26919,-3618
C06260=7394,30130,-30937,162,-26919,-3623
C06261=7407,30132,-30935,160,-26920,-3628
C06262=7419,30128,-30939,158,-26919,-3632
C06263=7430,30126,-30943,157,-26918,-3637
C06264=7443,30128,-30940,155,-26919,-3642
C06265=7454,30122,-30947,153,-26917,-3646
C06266=7464,30115,-30956,152,-26914,-3650
C06267=7460,30111,-30961,152,-26913,-3648
C06268=7448,30109,-30963,154,-26912,-3643
C06269=7437,30116,-30954,156,-26914,-3639
C06270=7425,30115,-30955,158,-26914,-3635
C06271=7412,30113,-30958,159,-26913,-3630
C06272=7399,30112,-30960,161,-26913,-3625
C06273=7386,30110,-30962,163,-26912,-3620
C06274=7373,30108,-30964,165,-26911,-3615
C06275=7363,30115,-30956,167,-26914,-3611
C06276=7350,30114,-30957,169,-26913,-3606
C06277=7337,30112,-30959,170,-26912,-3601
C06278=7326,30115,-30956,172,-26913,-3596
C06279=7314,30119,-30952,174,-26915,-3592
C06280=7303,30122,-30948,176,-26916,-3588
C06281=7292,30125,-30944,177,-26917,-3583
C06282=7280,30129,-30940,179,-26918,-3579
C06283=7269,30131,-30937,181,-26919,-3574
C06284=7258,30135,-30931,182,-26921,-3570
C06285=7246,30137,-30929,184,-26921,-3566
C06286=7235,30142,-30923,186,-26923,-3561
C06287=7225,30149,-30915,187,-26925,-3557
C06288=7213,30152,-30912,189,-26926,-3553
C06289=7202,30156,-30907,190,-26928,-3548
C06290=7192,30163,-30898,192,-26930,-3544
C06291=7180,30166,-30894,194,-26932,-3540
C06292=7169,30170,-30890,195,-26933,-3536
C06293=7157,30173,-30887,197,-26934,-3531
C06294=7146,30177,-30882,198,-26935,-3527
C06295=7134,30179,-30879,200,-26936,-3522
C06296=7130,30187,-30869,201,-26939,-3521
C06297=7130,30197,-29457,201,-26943,-3521
C06298=-41004,59868,4099,4900,-34257,16705
C06299=-41004,59868,1099,4900,-34257,16705
C06300=-41004,64596,1380,5213,-31659,16463
C06301=-41004,59868,1099,4900,-34257,16705
C06302=-41004,59868,9099,4900,-34257,16705
C06303=7130,30197,-26857,201,-26943,-3521
C06304=7130,30197,-30857,201,-26943,-3521
C06305=7130,30197,-29457,201,-26943,-3521
C06306=7101,30375,-26641,204,-27009,-3509
C06307=7101,30375,-30641,204,-27009,-3509
C06308=7101,30386,-30628,204,-27013,-3509
C06309=7108,30395,-30617,203,-27017,-3512
C06310=7119,30397,-30614,201,-27018,-3516
C06311=7131,30399,-30612,200,-27018,-3520
C06312=7142,30402,-30608,198,-27020,-3524
C06313=7149,30411,-30597,197,-27023,-3527
C06314=7161,30413,-30595,195,-27024,-3532
C06315=7172,30414,-30593,194,-27024,-3536
C06316=7184,30416,-30591,192,-27025,-3541
C06317=7193,30422,-30584,190,-27027,-3544
C06318=7202,30428,-30576,189,-27030,-3548
C06319=7214,30430,-30574,187,-27031,-3552
C06320=7226,30432,-30572,186,-27031,-3557
C06321=7237,30433,-30570,184,-27032,-3561
C06322=7249,30435,-30568,182,-27033,-3566
C06323=7261,30437,-30565,180,-27034,-3570
C06324=7268,30446,-30554,179,-27037,-3573
C06325=7279,30449,-30551,178,-27038,-3577
C06326=7291,30451,-30549,176,-27039,-3582
C06327=7302,30452,-30547,174,-27040,-3586
C06328=7314,30454,-30545,173,-27040,-3591
C06329=7326,30456,-30542,171,-27041,-3596
C06330=7338,30457,-30540,169,-27042,-3600
C06331=7349,30459,-30538,167,-27042,-3605
C06332=7361,30461,-30536,166,-27043,-3609
C06333=7373,30463,-30534,164,-27044,-3614
C06334=7385,30464,-30532,162,-27045,-3618
C06335=7396,30466,-30530,160,-27045,-3623
C06336=7408,30468,-30528,159,-27046,-3627
C06337=7419,30464,-30532,157,-27045,-3631
C06338=7420,30460,-30537,157,-27043,-3632
C06339=7408,30458,-30539,159,-27043,-3627
C06340=7396,30456,-30541,160,-27042,-3623
C06341=7385,30455,-30543,162,-27041,-3618
C06342=7377,30447,-30553,163,-27038,-3615
C06343=7367,30442,-30558,165,-27036,-3611
C06344=7355,30441,-30560,167,-27036,-3607
C06345=7343,30439,-30563,168,-27035,-3602
C06346=7331,30437,-30565,170,-27034,-3598
C06347=7320,30436,-30567,172,-27033,-3593
C06348=7308,30434,-30569,173,-27033,-3589
C06349=7299,30428,-30576,175,-27031,-3585
C06350=7290,30422,-30584,176,-27028,-3582
C06351=7278,30420,-30586,178,-27027,-3577
C06352=7267,30418,-30588,180,-27027,-3573
C06353=7255,30417,-30590,181,-27026,-3568
C06354=7243,30415,-30592,183,-27025,-3564
C06355=7232,30413,-30595,185,-27024,-3559
C06356=7224,30404,-30606,186,-27021,-3556
C06357=7213,30401,-30609,188,-27020,-3552
C06358=7202,30399,-30611,189,-27019,-3548
C06359=7190,30398,-30613,191,-27018,-3543
C06360=7180,30394,-30618,193,-27017,-3539
C06361=7172,30386,-30628,194,-27014,-3536
C06362=7160,30384,-30630,195,-27013,-3532
C06363=7148,30382,-30632,197,-27012,-3527
C06364=7137,30380,-30634,199,-27011,-3523
C06365=7125,30379,-30637,201,-27011,-3518
C06366=7113,30377,-30639,202,-27010,-3514
C06367=7101,30375,-30641,204,-27009,-3509
C06368=7101,30375,-29241,204,-27009,-3509
C06369=6246,30194,-26864,331,-26935,-3179
C06370=6246,30194,-30864,331,-26935,-3179
C06371=6234,30183,-30878,333,-26931,-3175
C06372=6211,30180,-30882,337,-26930,-3166
C06373=6192,30188,-30871,339,-26933,-3158
C06374=6175,30186,-30874,342,-26932,-3152
C06375=6153,30181,-30880,345,-26930,-3143
C06376=6135,30170,-30894,348,-26925,-3136
C06377=6113,30165,-30899,351,-26924,-3128
C06378=6090,30164,-30901,354,-26923,-3119
C06379=6070,30169,-30895,357,-26925,-3111
C06380=6046,30165,-30900,361,-26923,-3102
C06381=6023,30162,-30904,364,-26922,-3093
C06382=6004,30153,-30914,367,-26918,-3086
C06383=5983,30147,-30923,370,-26916,-3078
C06384=5960,30143,-30927,374,-26914,-3069
C06385=5937,30140,-30931,377,-26913,-3060
C06386=5913,30137,-30935,381,-26911,-3051
C06387=5890,30133,-30939,384,-26910,-3042
C06388=5867,30130,-30943,387,-26909,-3033
C06389=5844,30127,-30947,391,-26907,-3024
C06390=5827,30115,-30962,394,-26903,-3017
C06391=5804,30111,-30966,397,-26901,-3008
C06392=5780,30108,-30970,400,-26900,-3000
C06393=5757,30104,-30975,404,-26898,-2991
C06394=5734,30101,-30979,407,-26897,-2982
C06395=5711,30098,-30983,411,-26895,-2973
C06396=5688,30094,-30987,414,-26894,-2964
C06397=5668,30087,-30996,417,-26891,-2956
C06398=5647,30079,-31006,420,-26888,-2948
C06399=5624,30076,-31010,424,-26887,-2939
C06400=5601,30072,-31014,427,-26885,-2930
C06401=5610,30075,-31011,426,-26886,-2934
C06402=5629,30083,-31000,423,-26889,-2941
C06403=5645,30098,-30983,420,-26895,-2947
C06404=5668,30101,-30979,417,-26896,-2956
C06405=5691,30104,-30975,414,-26898,-2965
C06406=5709,30117,-30960,411,-26902,-2972
C06407=5732,30120,-30956,408,-26904,-2981
C06408=5755,30123,-30952,404,-26905,-2990
C06409=5778,30127,-30948,401,-26907,-2998
C06410=5801,30130,-30944,397,-26908,-3007
C06411=5824,30133,-30939,394,-26909,-3016
C06412=5847,30137,-30935,390,-26911,-3025
C06413=5870,30140,-30931,387,-26912,-3034
C06414=5893,30143,-30927,384,-26914,-3043
C06415=5911,30155,-30912,381,-26918,-3050
C06416=5934,30159,-30908,377,-26920,-3059
C06417=5957,30162,-30904,374,-26921,-3068
C06418=5980,30165,-30900,371,-26923,-3076
C06419=6003,30169,-30896,367,-26924,-3085
C06420=6021,30181,-30881,365,-26929,-3092
C06421=6044,30184,-30877,361,-26930,-3101
C06422=6067,30187,-30873,358,-26932,-3110
C06423=6090,30191,-30869,354,-26933,-3119
C06424=6113,30194,-30864,351,-26934,-3128
C06425=6136,30197,-30860,347,-26936,-3137
C06426=6159,30201,-30856,344,-26937,-3146
C06427=6182,30203,-30853,341,-26938,-3154
C06428=6202,30197,-30860,338,-26936,-3162
C06429=6226,30201,-30856,334,-26938,-3171
C06430=6246,30194,-30864,331,-26935,-3179
C06431=6246,30194,-29464,331,-26935,-3179
C06432=6235,30039,-27052,334,-26877,-3176
C06433=6235,30039,-31052,334,-26877,-3176
C06434=6254,30035,-31057,331,-26876,-3183
C06435=6243,30026,-31067,333,-26873,-3179
C06436=6225,30019,-31077,335,-26870,-3171
C06437=6203,30016,-31081,339,-26868,-3163
C06438=6188,30004,-31095,341,-26864,-3157
C06439=6166,30001,-31099,344,-26862,-3149
C06440=6150,29990,-31111,347,-26859,-3143
C06441=6129,29986,-31117,350,-26857,-3135
C06442=6108,29983,-31121,353,-26855,-3127
C06443=6087,29980,-31125,356,-26854,-3118
C06444=6069,29970,-31136,359,-26850,-3112
C06445=6050,29965,-31143,362,-26848,-3104
C06446=6029,29962,-31147,365,-26847,-3096
C06447=6007,29959,-31150,368,-26846,-3088
C06448=5986,29955,-31154,371,-26844,-3080
C06449=5965,29952,-31158,374,-26843,-3071
C06450=5943,29949,-31162,377,-26842,-3063
C06451=5922,29946,-31166,381,-26840,-3055
C06452=5904,29953,-31157,383,-26843,-3048
C06453=5883,29950,-31161,386,-26842,-3040
C06454=5864,29957,-31153,389,-26844,-3033
C06455=5843,29954,-31157,392,-26843,-3024
C06456=5823,29954,-31156,395,-26843,-3017
C06457=5804,29958,-31152,398,-26844,-3009
C06458=5785,29963,-31146,401,-26846,-3002
C06459=5764,29962,-31148,404,-26845,-2994
C06460=5746,29969,-31139,406,-26847,-2987
C06461=5726,29969,-31138,409,-26848,-2979
C06462=5707,29974,-31133,412,-26849,-2972
C06463=5688,29980,-31126,415,-26851,-2964
C06464=5667,29976,-31130,418,-26850,-2956
C06465=5675,29987,-31117,417,-26854,-2959
C06466=5694,29983,-31122,414,-26852,-2967
C06467=5714,29983,-31122,411,-26853,-2974
C06468=5735,29986,-31118,408,-26854,-2983
C06469=5754,29979,-31126,405,-26852,-2990
C06470=5775,29982,-31122,402,-26853,-2998
C06471=5793,29976,-31131,399,-26850,-3005
C06472=5814,29978,-31128,396,-26851,-3013
C06473=5833,29972,-29735,394,-26849,-3020
C06474=-41004,59868,4099,4900,-34257,16705
C06475=-41004,59868,1099,4900,-34257,16705
C06476=-41004,64596,1380,5213,-31659,16463
C06477=-41004,59868,1099,4900,-34257,16705
C06478=-41004,59868,9099,4900,-34257,16705
C06479=5833,29972,-27135,394,-26849,-3020
C06480=5833,29972,-31135,394,-26849,-3020
C06481=5854,29975,-31131,390,-26851,-3028
C06482=5872,29968,-31140,388,-26848,-3036
C06483=5893,29971,-31136,385,-26849,-3044
C06484=5912,29964,-31144,382,-26847,-3051
C06485=5933,29967,-31141,379,-26848,-3059
C06486=5954,29970,-31137,376,-26849,-3067
C06487=5975,29973,-31133,373,-26851,-3075
C06488=5997,29976,-31129,369,-26852,-3084
C06489=6018,29979,-31125,366,-26853,-3092
C06490=6039,29982,-31122,363,-26855,-3100
C06491=6060,29985,-31118,360,-26856,-3108
C06492=6079,29993,-31109,357,-26859,-3115
C06493=6097,30000,-31100,354,-26862,-3122
C06494=6119,30003,-31096,351,-26863,-3131
C06495=6140,30006,-31092,348,-26864,-3139
C06496=6156,30018,-31078,346,-26869,-3145
C06497=6177,30021,-31074,342,-26870,-3153
C06498=6197,30026,-31068,339,-26872,-3161
C06499=6214,30036,-31055,337,-26876,-3167
C06500=6235,30039,-31052,334,-26877,-3176
C06501=6235,30039,-29652,334,-26877,-3176
C06502=5942,29624,-27557,380,-26720,-3064
C06503=5942,29624,-31557,380,-26720,-3064
C06504=5950,29620,-31561,378,-26719,-3067
C06505=5954,29616,-31566,378,-26717,-3069
C06506=5945,29614,-31568,379,-26717,-3065
C06507=5936,29613,-31570,381,-26716,-3062
C06508=5930,29607,-31577,382,-26714,-3059
C06509=5924,29602,-31583,382,-26712,-3057
C06510=5915,29600,-31585,384,-26711,-3054
C06511=5906,29599,-31587,385,-26711,-3050
C06512=5897,29598,-31588,386,-26710,-3047
C06513=5888,29597,-31590,388,-26710,-3043
C06514=5879,29595,-31591,389,-26709,-3040
C06515=5870,29594,-31593,391,-26708,-3036
C06516=5861,29593,-31595,392,-26708,-3033
C06517=5852,29591,-31596,393,-26707,-3029
C06518=5843,29590,-31598,395,-26707,-3026
C06519=5834,29589,-31599,396,-26706,-3022
C06520=5825,29588,-31601,397,-26706,-3019
C06521=5818,29583,-31607,398,-26704,-3016
C06522=5813,29576,-31615,399,-26701,-3014
C06523=5804,29575,-31616,400,-26701,-3011
C06524=5795,29574,-31618,402,-26700,-3007
C06525=5786,29572,-31620,403,-26700,-3004
C06526=5777,29571,-31621,404,-26699,-3000
C06527=5768,29570,-31623,406,-26699,-2997
C06528=5760,29567,-31626,407,-26698,-2994
C06529=5754,29560,-31634,408,-26695,-2992
C06530=5746,29557,-31638,409,-26694,-2989
C06531=5738,29556,-31640,410,-26693,-2985
C06532=5729,29554,-31641,412,-26693,-2982
C06533=5720,29553,-31643,413,-26692,-2978
C06534=5711,29552,-31645,414,-26692,-2975
C06535=5710,29560,-31635,414,-26695,-2975
C06536=5717,29562,-31632,413,-26696,-2977
C06537=5724,29567,-31626,412,-26698,-2980
C06538=5729,29574,-31618,411,-26700,-2982
C06539=5738,29575,-31616,410,-26701,-2986
C06540=5747,29576,-31615,409,-26701,-2989
C06541=5756,29578,-31613,407,-26702,-2992
C06542=5765,29579,-31612,406,-26702,-2996
C06543=5774,29580,-31610,405,-26703,-2999
C06544=5782,29583,-31607,404,-26704,-3002
C06545=5788,29590,-31599,403,-26706,-3005
C06546=5796,29593,-31595,402,-26708,-3008
C06547=5805,29594,-31593,400,-26708,-3011
C06548=5814,29595,-31591,399,-26709,-3015
C06549=5822,29597,-31590,398,-26709,-3018
C06550=5831,29598,-31588,396,-26710,-3021
C06551=5840,29599,-31587,395,-26710,-3025
C06552=5849,29601,-31585,394,-26711,-3028
C06553=5858,29602,-31583,392,-26711,-3032
C06554=5867,29603,-31582,391,-26712,-3035
C06555=5876,29604,-31580,389,-26712,-3039
C06556=5885,29606,-31579,388,-26713,-3042
C06557=5894,29607,-31577,387,-26714,-3045
C06558=5900,29614,-31568,386,-26716,-3048
C06559=5907,29618,-31563,385,-26718,-3050
C06560=5916,29620,-31562,384,-26718,-3054
C06561=5925,29621,-31560,382,-26719,-3057
C06562=5934,29622,-31558,381,-26719,-3061
C06563=5942,29624,-31557,380,-26720,-3064
C06564=5942,29624,-30157,380,-26720,-3064
C06565=5325,29516,-27690,472,-26676,-2826
C06566=5325,29516,-31690,472,-26676,-2826
C06567=5322,29450,-31769,473,-26651,-2825
C06568=5323,29384,-31849,473,-26627,-2826
C06569=5315,29321,-31926,475,-26603,-2823
C06570=5293,29260,-32000,478,-26580,-2815
C06571=5275,29198,-32075,481,-26557,-2808
C06572=5266,29134,-32152,483,-26533,-2805
C06573=5258,29070,-32230,485,-26509,-2803
C06574=5257,29005,-32309,486,-26485,-2803
C06575=5256,28939,-32389,486,-26460,-2803
C06576=5247,28875,-32466,488,-26436,-2799
C06577=5253,28808,-32547,488,-26411,-2802
C06578=5250,28743,-32626,489,-26387,-2801
C06579=5245,28678,-32704,490,-26363,-2799
C06580=5233,28615,-32781,492,-26339,-2795
C06581=5219,28552,-32857,495,-26316,-2790
C06582=5195,28492,-32931,499,-26293,-2781
C06583=5170,28431,-33004,503,-26271,-2772
C06584=5146,28371,-33077,507,-26248,-2763
C06585=5129,28308,-33153,510,-26225,-2757
C06586=5106,28247,-33227,514,-26202,-2748
C06587=5081,28187,-33300,518,-26179,-2739
C06588=5056,28127,-33373,522,-26157,-2730
C06589=5031,28066,-33446,527,-26134,-2720
C06590=4998,28007,-33518,532,-26112,-2708
C06591=4966,27948,-33589,537,-26090,-2696
C06592=4922,27897,-33651,544,-26070,-2679
C06593=4954,27956,-33580,539,-26093,-2691
C06594=4987,28015,-33508,534,-26115,-2704
C06595=5019,28074,-33437,528,-26137,-2716
C06596=5044,28135,-33364,524,-26159,-2725
C06597=5069,28195,-33290,520,-26182,-2734
C06598=5085,28257,-33215,517,-26205,-2740
C06599=5109,28318,-33141,513,-26228,-2749
C06600=5122,28381,-33065,510,-26252,-2754
C06601=5136,28444,-32989,508,-26275,-2759
C06602=5161,28504,-32915,504,-26298,-2768
C06603=5186,28565,-32842,499,-26320,-2777
C06604=5209,28626,-32768,496,-26343,-2786
C06605=5224,28688,-32693,493,-26367,-2792
C06606=5227,28753,-32614,492,-26391,-2792
C06607=5230,28818,-32535,491,-26415,-2793
C06608=5222,28886,-32453,492,-26440,-2790
C06609=5224,28951,-32374,491,-26465,-2790
C06610=5227,29016,-32295,490,-26489,-2791
C06611=5230,29082,-32216,489,-26513,-2792
C06612=5232,29147,-32137,488,-26537,-2792
C06613=5246,29210,-32061,486,-26561,-2797
C06614=5264,29271,-31986,483,-26584,-2804
C06615=5280,29334,-31910,480,-26607,-2810
C06616=5289,29397,-31833,478,-26631,-2813
C06617=5300,29461,-31756,476,-26655,-2817
C06618=5291,29528,-31674,477,-26680,-2813
C06619=5273,29591,-31599,479,-26703,-2806
C06620=5245,29647,-31530,483,-26724,-2795
C06621=5222,29707,-31459,486,-26746,-2785
C06622=5223,29749,-31408,485,-26762,-2786
C06623=5250,29691,-31477,482,-26741,-2796
C06624=5277,29634,-31546,478,-26719,-2807
C06625=5306,29578,-31614,474,-26699,-2819
C06626=5325,29516,-31690,472,-26676,-2826
C06627=5325,29516,-30290,472,-26676,-2826
C06628=5134,29520,-27686,500,-26676,-2753
C06629=5134,29520,-31686,500,-26676,-2753
C06630=5143,29444,-31777,499,-26648,-2756
C06631=5124,29375,-31861,502,-26622,-2749
C06632=5107,29306,-31945,506,-26596,-2743
C06633=5095,29235,-32031,508,-26569,-2739
C06634=5070,29172,-32106,512,-26546,-2730
C06635=5072,29245,-32018,511,-26573,-2730
C06636=5085,29316,-31933,509,-26599,-2735
C06637=5108,29384,-31850,505,-26625,-2743
C06638=5121,29455,-31764,502,-26651,-2748
C06639=5107,29527,-31677,504,-26678,-2742
C06640=5073,29589,-31602,508,-26701,-2729
C06641=5044,29654,-31524,512,-26725,-2717
C06642=5016,29718,-31445,516,-26749,-2706
C06643=5006,29794,-31354,517,-26777,-2702
C06644=5019,29864,-31269,514,-26803,-2706
C06645=5053,29930,-31189,509,-26828,-2719
C06646=5076,29998,-31106,505,-26853,-2728
C06647=5089,30068,-31021,503,-26880,-2732
C06648=5079,30144,-30930,503,-26908,-2728
C06649=5060,30214,-29445,506,-26934,-2721
C06650=-41004,59868,4099,4900,-34257,16705
C06651=-41004,59868,1099,4900,-34257,16705
C06652=-41004,64596,1380,5213,-31659,16463
C06653=-41004,59868,1099,4900,-34257,16705
C06654=-41004,59868,9099,4900,-34257,16705
C06655=5060,30214,-26845,506,-26934,-2721
C06656=5060,30214,-30845,506,-26934,-2721
C06657=5024,30274,-30772,511,-26956,-2706
C06658=4987,30334,-30699,516,-26978,-2692
C06659=4965,30402,-30617,518,-27003,-2683
C06660=4966,30475,-30529,518,-27030,-2683
C06661=4968,30548,-30440,517,-27058,-2683
C06662=4969,30621,-30352,516,-27085,-2683
C06663=4960,30696,-30261,517,-27113,-2679
C06664=4932,30761,-30183,521,-27137,-2668
C06665=4902,30825,-30106,524,-27160,-2656
C06666=4885,30895,-30020,526,-27186,-2649
C06667=4889,30968,-29932,525,-27213,-2651
C06668=4888,31041,-29843,525,-27241,-2650
C06669=4859,31106,-29765,529,-27265,-2638
C06670=4831,31170,-29687,532,-27288,-2627
C06671=4826,31209,-29640,533,-27303,-2625
C06672=4859,31147,-29715,528,-27280,-2638
C06673=4893,31085,-29790,524,-27257,-2651
C06674=4911,31015,-29875,522,-27231,-2659
C06675=4899,30945,-29960,524,-27205,-2655
C06676=4898,30872,-30048,525,-27178,-2654
C06677=4926,30807,-30126,521,-27154,-2666
C06678=4955,30743,-30205,517,-27130,-2677
C06679=4974,30673,-30289,515,-27104,-2685
C06680=4992,30603,-30374,513,-27078,-2692
C06681=4980,30532,-30459,515,-27052,-2688
C06682=4979,30459,-30548,516,-27025,-2688
C06683=4988,30384,-30639,515,-26997,-2692
C06684=5016,30319,-30717,511,-26973,-2703
C06685=5055,30260,-30789,506,-26951,-2718
C06686=5093,30201,-30861,501,-26929,-2733
C06687=5112,30131,-30945,499,-26903,-2741
C06688=5111,30058,-31033,499,-26876,-2741
C06689=5098,29988,-31119,502,-26850,-2736
C06690=5075,29919,-31201,506,-26824,-2728
C06691=5046,29853,-31282,510,-26799,-2717
C06692=5029,29783,-31367,514,-26773,-2710
C06693=5048,29713,-31451,511,-26747,-2718
C06694=5067,29643,-31536,509,-26721,-2726
C06695=5102,29582,-31610,504,-26699,-2740
C06696=5134,29520,-31686,500,-26676,-2753
C06697=5134,29520,-30286,500,-26676,-2753
C06698=4740,29379,-27857,559,-26621,-2601
C06699=4740,29379,-31857,559,-26621,-2601
C06700=4670,29491,-31721,569,-26662,-2573
C06701=4578,29591,-31601,581,-26698,-2538
C06702=4478,29686,-31487,596,-26733,-2498
C06703=4357,29770,-31386,613,-26763,-2451
C06704=4228,29825,-31319,631,-26783,-2401
C06705=4094,29864,-31273,651,-26796,-2349
C06706=3952,29880,-31254,671,-26801,-2294
C06707=3806,29880,-31255,693,-26800,-2237
C06708=3697,29845,-31297,709,-26786,-2195
C06709=3556,29801,-31351,730,-26769,-2141
C06710=3446,29704,-31469,747,-26732,-2099
C06711=3347,29588,-31609,763,-26688,-2061
C06712=3254,29471,-31751,778,-26644,-2027
C06713=3192,29347,-31902,788,-26598,-2003
C06714=3145,29219,-32056,796,-26550,-1986
C06715=3105,29090,-32213,804,-26502,-1972
C06716=3086,28956,-32375,808,-26452,-1965
C06717=3077,28819,-32540,811,-26402,-1963
C06718=3079,28681,-32708,812,-26350,-1964
C06719=3092,28539,-32879,811,-26298,-1970
C06720=3125,28409,-33036,808,-26250,-1984
C06721=3226,28342,-33116,794,-26226,-2023
C06722=3372,28335,-33125,772,-26224,-2080
C06723=3514,28367,-33086,750,-26237,-2134
C06724=3619,28466,-32966,734,-26274,-2174
C06725=3627,28602,-32801,731,-26325,-2176
C06726=3613,28743,-32631,732,-26377,-2170
C06727=3621,28790,-32574,730,-26394,-2173
C06728=3643,28654,-32739,728,-26344,-2182
C06729=3647,28515,-32907,729,-26292,-2184
C06730=3581,28391,-33056,740,-26246,-2160
C06731=3449,28327,-33135,760,-26221,-2110
C06732=3296,28314,-33150,783,-26216,-2050
C06733=3153,28333,-33128,804,-26222,-1995
C06734=3132,28216,-33270,809,-26178,-1988
C06735=3145,28074,-33440,808,-26126,-1994
C06736=3168,27939,-33605,806,-26076,-2004
C06737=3212,27814,-33756,801,-26030,-2022
C06738=3276,27700,-33893,793,-25988,-2047
C06739=3391,27629,-33978,776,-25963,-2092
C06740=3532,27602,-34010,755,-25953,-2146
C06741=3680,27595,-34019,733,-25951,-2204
C06742=3825,27577,-34040,712,-25946,-2259
C06743=3975,27599,-34014,689,-25955,-2317
C06744=4124,27639,-33965,666,-25970,-2374
C06745=4270,27682,-33912,644,-25987,-2430
C06746=4402,27748,-33832,624,-26012,-2480
C06747=4511,27852,-33707,606,-26051,-2522
C06748=4597,27971,-33563,592,-26096,-2554
C06749=4689,28088,-33420,578,-26140,-2589
C06750=4798,28191,-33295,560,-26179,-2630
C06751=4841,28319,-33140,553,-26227,-2646
C06752=4822,28459,-32971,555,-26279,-2638
C06753=4809,28593,-32808,555,-26329,-2632
C06754=4836,28725,-32649,550,-26378,-2642
C06755=4835,28849,-32499,549,-26424,-2641
C06756=4791,28975,-32347,555,-26471,-2623
C06757=4750,29102,-32192,560,-26518,-2607
C06758=4734,29243,-32022,561,-26570,-2600
C06759=4740,29379,-31857,559,-26621,-2601
C06760=4740,29379,-30457,559,-26621,-2601
C06761=5067,29097,-28197,513,-26518,-2729
C06762=5067,29097,-32197,513,-26518,-2729
C06763=5082,29079,-32220,511,-26511,-2735
C06764=5095,29059,-32244,509,-26504,-2740
C06765=5098,29034,-32274,509,-26495,-2741
C06766=5111,29014,-32298,507,-26487,-2746
C06767=5114,28989,-32328,507,-26478,-2747
C06768=5127,28970,-32352,505,-26471,-2752
C06769=5130,28945,-32382,505,-26462,-2754
C06770=5133,28920,-32412,505,-26452,-2755
C06771=5136,28895,-32443,504,-26443,-2756
C06772=5139,28870,-32473,504,-26434,-2758
C06773=5131,28847,-32501,505,-26425,-2755
C06774=5134,28822,-32531,505,-26416,-2756
C06775=5127,28799,-32559,506,-26407,-2754
C06776=5125,28775,-32588,507,-26398,-2753
C06777=5121,28752,-32616,508,-26390,-2751
C06778=5113,28729,-32643,509,-26381,-2748
C06779=5103,28707,-32670,511,-26373,-2745
C06780=5093,28684,-32697,512,-26364,-2741
C06781=5084,28662,-32724,514,-26356,-2737
C06782=5074,28640,-32751,516,-26348,-2734
C06783=5064,28618,-32778,517,-26339,-2730
C06784=5054,28595,-32805,519,-26331,-2726
C06785=5046,28573,-32833,520,-26323,-2724
C06786=5038,28550,-32860,522,-26314,-2721
C06787=5030,28528,-32888,523,-26306,-2718
C06788=5022,28505,-32915,524,-26297,-2715
C06789=5014,28482,-32942,526,-26289,-2712
C06790=5006,28460,-32970,527,-26280,-2709
C06791=4998,28437,-32997,529,-26272,-2706
C06792=4978,28422,-33015,532,-26266,-2698
C06793=4987,28445,-32988,530,-26275,-2701
C06794=4995,28467,-32960,529,-26283,-2704
C06795=5003,28490,-32933,527,-26292,-2707
C06796=5011,28513,-32905,526,-26300,-2710
C06797=5019,28535,-32878,525,-26308,-2713
C06798=5027,28558,-32851,523,-26317,-2716
C06799=5032,28581,-32823,522,-26326,-2718
C06800=5042,28603,-32796,521,-26334,-2722
C06801=5051,28626,-32768,519,-26342,-2725
C06802=5059,28649,-32741,518,-26351,-2728
C06803=5067,28671,-32713,516,-26359,-2731
C06804=5074,28694,-32686,515,-26368,-2734
C06805=5082,28717,-32658,514,-26376,-2737
C06806=5090,28739,-32631,512,-26385,-2740
C06807=5098,28762,-32604,511,-26393,-2743
C06808=5106,28785,-32576,510,-26402,-2746
C06809=5114,28807,-32549,508,-26410,-2749
C06810=5111,28832,-32518,509,-26420,-2747
C06811=5119,28855,-32491,507,-26428,-2750
C06812=5116,28880,-32461,507,-26437,-2749
C06813=5113,28905,-32430,508,-26447,-2748
C06814=5110,28930,-32400,508,-26456,-2746
C06815=5107,28955,-32370,508,-26465,-2745
C06816=5104,28980,-32339,508,-26475,-2744
C06817=5094,29001,-32314,510,-26482,-2740
C06818=5088,29025,-32285,510,-26491,-2737
C06819=5075,29044,-32262,512,-26498,-2732
C06820=5064,29065,-32237,514,-26506,-2728
C06821=5059,29089,-32207,514,-26515,-2726
C06822=5067,29097,-30797,513,-26518,-2729
C06823=-41004,59868,4099,4900,-34257,16705
C06824=-41004,59868,1099,4900,-34257,16705
C06825=-41004,64596,1380,5213,-31659,16463
C06826=-41004,59868,1099,4900,-34257,16705
C06827=-41004,59868,9099,4900,-34257,16705
C06828=5067,29097,-28197,513,-26518,-2729
C06829=5067,29097,-32197,513,-26518,-2729
C06830=5067,29097,-30797,513,-26518,-2729
C06831=5651,28863,-28479,428,-26434,-2955
C06832=5651,28863,-32479,428,-26434,-2955
C06833=5661,28875,-32466,426,-26439,-2959
C06834=5679,28886,-32452,424,-26443,-2966
C06835=5701,28890,-32447,420,-26445,-2974
C06836=5724,28893,-32443,417,-26446,-2983
C06837=5741,28905,-32429,414,-26451,-2990
C06838=5763,28908,-32424,411,-26452,-2998
C06839=5786,28912,-32420,408,-26453,-3007
C06840=5809,28915,-32416,404,-26455,-3016
C06841=5831,28918,-32412,401,-26456,-3024
C06842=5848,28930,-32398,398,-26461,-3031
C06843=5865,28943,-32382,396,-26465,-3037
C06844=5879,28959,-32362,393,-26472,-3043
C06845=5897,28970,-32350,391,-26476,-3049
C06846=5911,28986,-32329,388,-26482,-3055
C06847=5928,28999,-32314,386,-26487,-3061
C06848=5943,29014,-32296,383,-26492,-3067
C06849=5957,29030,-32276,381,-26499,-3072
C06850=5971,29047,-32256,379,-26505,-3078
C06851=5989,29057,-32243,376,-26509,-3085
C06852=6003,29074,-32223,374,-26515,-3090
C06853=6017,29091,-32203,372,-26521,-3095
C06854=6031,29107,-32183,370,-26528,-3101
C06855=6047,29122,-32165,367,-26533,-3107
C06856=6063,29134,-32150,365,-26538,-3113
C06857=6081,29146,-32136,362,-26542,-3120
C06858=6098,29158,-32121,359,-26547,-3126
C06859=6115,29170,-32107,357,-26552,-3132
C06860=6132,29182,-32092,354,-26556,-3139
C06861=6153,29186,-32086,351,-26558,-3147
C06862=6169,29190,-32082,349,-26559,-3153
C06863=6166,29177,-32098,349,-26555,-3152
C06864=6149,29165,-32112,352,-26550,-3146
C06865=6129,29158,-32121,355,-26547,-3138
C06866=6111,29147,-32134,358,-26543,-3131
C06867=6093,29137,-32147,360,-26539,-3124
C06868=6079,29120,-32167,363,-26533,-3119
C06869=6061,29110,-32180,365,-26529,-3112
C06870=6047,29093,-32200,367,-26523,-3107
C06871=6033,29076,-32220,370,-26516,-3101
C06872=6015,29066,-32233,372,-26512,-3095
C06873=6001,29049,-32253,375,-26506,-3089
C06874=5987,29033,-32273,377,-26500,-3084
C06875=5973,29016,-32293,379,-26493,-3078
C06876=5959,28999,-32314,381,-26487,-3073
C06877=5941,28989,-32326,384,-26483,-3066
C06878=5927,28972,-32346,386,-26477,-3061
C06879=5911,28958,-32363,389,-26471,-3055
C06880=5895,28945,-32379,391,-26467,-3049
C06881=5877,28934,-32393,394,-26462,-3042
C06882=5860,28922,-32407,396,-26458,-3035
C06883=5843,28910,-32422,399,-26453,-3029
C06884=5820,28907,-32426,402,-26452,-3020
C06885=5800,28899,-32435,405,-26449,-3013
C06886=5781,28892,-32445,408,-26446,-3005
C06887=5758,28888,-32449,412,-26444,-2996
C06888=5735,28885,-32453,415,-26443,-2988
C06889=5718,28873,-32467,418,-26439,-2981
C06890=5696,28870,-32471,421,-26437,-2972
C06891=5673,28867,-32475,425,-26436,-2964
C06892=5651,28863,-32479,428,-26434,-2955
C06893=5651,28863,-31079,428,-26434,-2955
C06894=6285,28904,-28428,333,-26454,-3199
C06895=6285,28904,-32428,333,-26454,-3199
C06896=6289,28912,-32419,333,-26456,-3201
C06897=6294,28919,-32411,332,-26459,-3203
C06898=6293,28927,-32400,332,-26462,-3202
C06899=6292,28936,-32390,332,-26465,-3202
C06900=6297,28943,-32381,331,-26468,-3204
C06901=6300,28950,-32372,331,-26471,-3205
C06902=6301,28958,-32362,330,-26474,-3205
C06903=6307,28965,-32354,330,-26477,-3207
C06904=6308,28973,-32344,329,-26480,-3208
C06905=6311,28981,-32335,329,-26482,-3209
C06906=6317,28988,-32326,328,-26485,-3211
C06907=6315,28997,-32316,328,-26488,-3211
C06908=6314,29005,-32306,328,-26491,-3210
C06909=6313,29014,-32296,328,-26495,-3210
C06910=6317,29021,-32286,328,-26497,-3211
C06911=6323,29028,-32278,327,-26500,-3213
C06912=6329,29035,-32270,326,-26503,-3216
C06913=6334,29042,-32261,325,-26505,-3218
C06914=6340,29049,-32253,324,-26508,-3220
C06915=6346,29056,-32244,323,-26511,-3222
C06916=6352,29063,-32236,322,-26513,-3224
C06917=6358,29070,-32227,321,-26516,-3227
C06918=6358,29078,-32217,321,-26519,-3227
C06919=6362,29085,-32208,321,-26522,-3228
C06920=6366,29093,-32199,320,-26524,-3230
C06921=6366,29100,-32190,320,-26527,-3230
C06922=6376,29102,-32188,318,-26528,-3233
C06923=6377,29093,-32199,318,-26525,-3234
C06924=6378,29085,-32209,318,-26522,-3234
C06925=6374,29078,-32218,319,-26519,-3233
C06926=6369,29070,-32227,320,-26516,-3231
C06927=6371,29062,-32237,319,-26513,-3232
C06928=6372,29053,-32247,319,-26510,-3232
C06929=6366,29046,-32256,320,-26507,-3230
C06930=6360,29039,-32264,321,-26504,-3228
C06931=6354,29032,-32273,322,-26502,-3225
C06932=6348,29025,-32281,323,-26499,-3223
C06933=6342,29018,-32290,324,-26497,-3221
C06934=6336,29011,-32298,325,-26494,-3219
C06935=6336,29003,-32308,325,-26491,-3218
C06936=6332,28996,-32317,326,-26488,-3217
C06937=6327,28989,-32326,326,-26485,-3215
C06938=6328,28980,-32336,326,-26482,-3216
C06939=6330,28972,-32346,326,-26479,-3216
C06940=6325,28965,-32355,327,-26476,-3214
C06941=6321,28957,-32364,327,-26474,-3213
C06942=6321,28949,-32374,328,-26470,-3213
C06943=6315,28942,-32382,329,-26468,-3211
C06944=6313,28934,-32392,329,-26465,-3210
C06945=6311,28926,-32401,329,-26462,-3209
C06946=6305,28919,-32410,330,-26459,-3207
C06947=6306,28911,-32420,330,-26456,-3207
C06948=6307,28902,-32430,330,-26453,-3208
C06949=6308,28894,-32441,330,-26450,-3208
C06950=6305,28886,-32450,330,-26447,-3207
C06951=6298,28880,-32458,331,-26445,-3205
C06952=6289,28879,-32459,333,-26444,-3201
C06953=6288,28887,-32449,333,-26447,-3200
C06954=6287,28896,-32439,333,-26450,-3200
C06955=6285,28904,-32428,333,-26454,-3199
C06956=6285,28904,-31028,333,-26454,-3199
C06957=5223,29829,-27310,485,-26792,-2785
C06958=5223,29829,-31310,485,-26792,-2785
C06959=5213,29825,-31316,486,-26790,-2781
C06960=5211,29837,-31301,486,-26795,-2781
C06961=5210,29850,-31285,486,-26799,-2780
C06962=5216,29860,-31272,485,-26803,-2782
C06963=5217,29872,-31258,485,-26808,-2783
C06964=5225,29883,-31245,484,-26812,-2786
C06965=5226,29895,-31231,484,-26816,-2786
C06966=5234,29905,-31218,482,-26820,-2789
C06967=5236,29917,-31204,482,-26824,-2790
C06968=5242,29927,-31191,481,-26828,-2792
C06969=5245,29939,-31177,480,-26833,-2793
C06970=5250,29950,-31164,480,-26837,-2795
C06971=5248,29963,-31149,480,-26842,-2794
C06972=5256,29973,-31136,479,-26846,-2797
C06973=5257,29985,-31121,478,-26850,-2798
C06974=5265,29995,-31109,477,-26854,-2801
C06975=5264,30008,-31094,477,-26859,-2800
C06976=5267,30019,-31080,477,-26863,-2801
C06977=5271,30030,-31066,476,-26867,-2803
C06978=5277,30041,-31053,475,-26871,-2805
C06979=5279,30053,-31039,475,-26875,-2806
C06980=5277,30065,-31024,475,-26880,-2805
C06981=5276,30078,-31009,475,-26885,-2805
C06982=5274,30090,-30994,475,-26889,-2804
C06983=5273,30103,-30978,475,-26894,-2803
C06984=5271,30115,-30963,475,-26899,-2803
C06985=5270,30128,-30948,476,-26903,-2802
C06986=5268,30140,-30933,476,-26908,-2801
C06987=5266,30153,-30918,476,-26913,-2801
C06988=5265,30165,-30903,476,-26917,-2800
C06989=5274,30161,-30908,475,-26916,-2803
C06990=5277,30150,-30922,474,-26912,-2805
C06991=5279,30137,-30937,474,-26907,-2805
C06992=5280,30125,-30952,474,-26902,-2806
C06993=5289,30116,-30962,473,-26899,-2809
C06994=5293,30105,-30976,472,-26895,-2811
C06995=5295,30092,-30991,472,-26890,-2812
C06996=5296,30080,-31006,472,-26886,-2813
C06997=5298,30067,-31021,472,-26881,-2813
C06998=5300,30055,-29636,472,-26876,-2814
C06999=-41004,59868,4099,4900,-34257,16705
C07000=-41004,59868,1099,4900,-34257,16705
C07001=-41004,64596,1380,5213,-31659,16463
C07002=-41004,59868,1099,4900,-34257,16705
C07003=-41004,59868,9099,4900,-34257,16705
C07004=5300,30055,-27036,472,-26876,-2814
C07005=5300,30055,-31036,472,-26876,-2814
C07006=5301,30043,-31051,471,-26872,-2814
C07007=5296,30032,-31065,472,-26868,-2812
C07008=5293,30020,-31079,473,-26863,-2812
C07009=5294,30008,-31094,473,-26859,-2812
C07010=5286,29997,-31106,474,-26855,-2809
C07011=5284,29986,-31121,474,-26850,-2808
C07012=5278,29975,-31134,475,-26846,-2806
C07013=5275,29963,-31147,476,-26842,-2805
C07014=5270,29952,-31161,477,-26838,-2803
C07015=5265,29941,-31174,477,-26834,-2801
C07016=5263,29930,-31188,478,-26829,-2800
C07017=5256,29919,-31201,479,-26825,-2798
C07018=5255,29907,-31216,479,-26821,-2797
C07019=5246,29897,-31228,481,-26817,-2794
C07020=5245,29885,-31243,481,-26813,-2794
C07021=5238,29874,-31255,482,-26809,-2791
C07022=5236,29863,-31269,482,-26804,-2790
C07023=5230,29852,-31283,483,-26800,-2788
C07024=5226,29841,-31296,484,-26796,-2786
C07025=5223,29829,-31310,485,-26792,-2785
C07026=5223,29829,-29910,485,-26792,-2785
C07027=5154,30218,-26839,492,-26936,-2757
C07028=5154,30218,-30839,492,-26936,-2757
C07029=5152,30231,-30824,492,-26941,-2756
C07030=5146,30241,-30812,493,-26945,-2754
C07031=5139,30251,-30800,494,-26948,-2751
C07032=5138,30264,-30784,494,-26953,-2750
C07033=5136,30276,-30769,494,-26958,-2750
C07034=5130,30286,-30757,495,-26961,-2747
C07035=5123,30296,-30745,496,-26965,-2745
C07036=5122,30309,-30729,496,-26970,-2744
C07037=5120,30322,-30714,496,-26975,-2743
C07038=5119,30334,-30698,496,-26979,-2743
C07039=5110,30343,-30688,497,-26982,-2739
C07040=5106,30354,-30674,498,-26987,-2737
C07041=5104,30367,-30659,498,-26991,-2737
C07042=5103,30380,-30644,498,-26996,-2736
C07043=5101,30392,-30628,498,-27001,-2735
C07044=5100,30405,-30613,498,-27005,-2735
C07045=5098,30418,-30597,499,-27010,-2734
C07046=5096,30431,-30582,499,-27015,-2733
C07047=5095,30443,-30567,499,-27020,-2733
C07048=5093,30456,-30551,499,-27024,-2732
C07049=5092,30469,-30536,499,-27029,-2732
C07050=5090,30481,-30521,499,-27034,-2731
C07051=5089,30494,-30505,499,-27039,-2730
C07052=5087,30507,-30490,500,-27043,-2730
C07053=5089,30519,-30475,499,-27048,-2730
C07054=5095,30530,-30462,498,-27052,-2732
C07055=5093,30542,-30447,498,-27057,-2732
C07056=5100,30553,-30433,497,-27061,-2734
C07057=5101,30564,-30420,497,-27065,-2735
C07058=5112,30557,-30429,496,-27062,-2739
C07059=5100,30553,-30434,497,-27060,-2734
C07060=5093,30542,-30447,498,-27056,-2732
C07061=5099,30531,-30460,498,-27053,-2734
C07062=5106,30522,-30471,497,-27049,-2737
C07063=5108,30509,-30487,497,-27044,-2737
C07064=5100,30499,-30500,498,-27040,-2734
C07065=5100,30486,-30515,498,-27036,-2735
C07066=5102,30473,-30530,498,-27031,-2735
C07067=5103,30461,-30545,498,-27026,-2736
C07068=5105,30448,-30561,497,-27021,-2737
C07069=5106,30435,-30576,497,-27017,-2737
C07070=5108,30423,-30592,497,-27012,-2738
C07071=5109,30410,-30607,497,-27007,-2739
C07072=5111,30397,-30622,497,-27003,-2739
C07073=5113,30385,-30638,497,-26998,-2740
C07074=5114,30372,-30653,497,-26993,-2741
C07075=5120,30362,-30665,496,-26989,-2743
C07076=5127,30352,-30677,495,-26986,-2746
C07077=5129,30339,-30693,495,-26981,-2746
C07078=5130,30326,-30708,495,-26976,-2747
C07079=5132,30314,-30723,494,-26972,-2748
C07080=5140,30305,-30734,493,-26968,-2751
C07081=5145,30294,-30748,493,-26964,-2753
C07082=5146,30281,-30763,493,-26960,-2753
C07083=5148,30268,-30778,492,-26955,-2754
C07084=5149,30256,-30794,492,-26950,-2755
C07085=5153,30244,-30807,492,-26946,-2756
C07086=5162,30236,-30818,491,-26943,-2760
C07087=5164,30223,-30833,490,-26938,-2760
C07088=5154,30218,-30839,492,-26936,-2757
C07089=5154,30218,-29439,492,-26936,-2757
C07090=5379,30277,-26767,458,-26960,-2843
C07091=5379,30277,-30767,458,-26960,-2843
C07092=5375,30289,-30753,459,-26964,-2842
C07093=5370,30300,-30739,459,-26968,-2840
C07094=5362,30309,-30728,461,-26972,-2837
C07095=5355,30319,-30716,462,-26975,-2834
C07096=5349,30330,-30703,462,-26979,-2832
C07097=5347,30343,-30687,463,-26984,-2831
C07098=5342,30354,-30674,463,-26988,-2829
C07099=5334,30363,-30663,464,-26992,-2826
C07100=5332,30376,-30647,465,-26996,-2825
C07101=5331,30389,-30631,465,-27001,-2824
C07102=5329,30402,-30616,465,-27006,-2824
C07103=5321,30411,-30604,466,-27010,-2821
C07104=5316,30423,-30591,467,-27014,-2819
C07105=5315,30435,-30575,467,-27018,-2818
C07106=5313,30448,-30559,467,-27023,-2817
C07107=5311,30461,-30544,467,-27028,-2816
C07108=5310,30474,-30528,467,-27033,-2816
C07109=5308,30487,-30512,467,-27038,-2815
C07110=5306,30500,-30497,467,-27043,-2814
C07111=5305,30513,-30481,468,-27047,-2814
C07112=5303,30526,-30465,468,-27052,-2813
C07113=5302,30539,-30450,468,-27057,-2812
C07114=5300,30552,-30434,468,-27062,-2812
C07115=5299,30564,-30419,468,-27066,-2811
C07116=5310,30557,-30428,467,-27064,-2815
C07117=5311,30544,-30444,466,-27059,-2816
C07118=5313,30531,-30460,466,-27054,-2817
C07119=5315,30518,-30475,466,-27049,-2818
C07120=5316,30505,-30491,466,-27044,-2818
C07121=5318,30492,-30507,466,-27040,-2819
C07122=5320,30479,-30522,466,-27035,-2820
C07123=5326,30468,-30535,465,-27031,-2822
C07124=5333,30458,-30547,464,-27027,-2825
C07125=5334,30446,-30563,464,-27022,-2825
C07126=5336,30433,-30579,464,-27018,-2826
C07127=5337,30420,-30594,464,-27013,-2827
C07128=5339,30407,-30610,463,-27008,-2827
